KUKA KRL program: EPS_2_25716_MHDR05_A_20250926070358.src

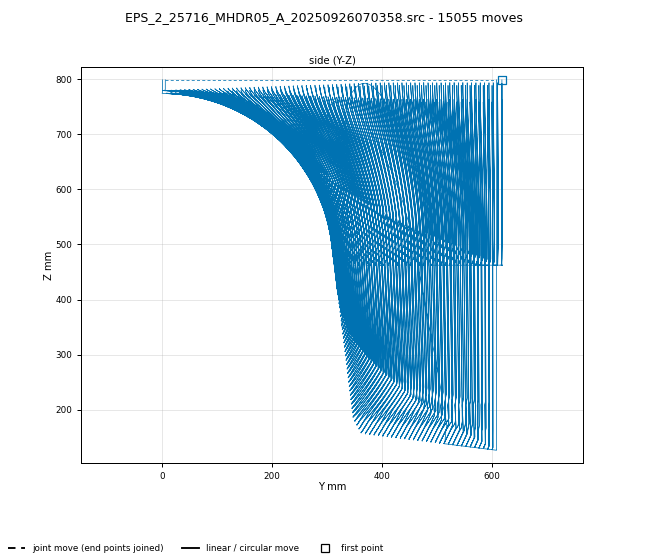
[picture p0: tool path of EPS_2_25716_MHDR05_A_20250926070358.src, 15055 of 15057 moves have a stored position in this frame; points joined in program order, loops and branches not executed]
&ACCESS RVP
&REL 4
&COMMENT QRS 19112012
&PARAM EDITMASK = *
DEF PART()
EXT BAS (BAS_COMMAND :IN,REAL :IN )
INT I
BAS (#INITMOV,0 )

;KUKA QRS Post kuka4.cps  Date:22-06-2017 !

File_ID=2854

QRS_PRE_INIT()

;Init var - Until changes are made in qrs_pre_init
Outlet_Square_prg=0
Inlet_1_Square_prg=0
Inlet_2_Square_prg=0
Inlet_3_Square_prg=0
Inlet_4_Square_prg=0
Inlet_5_Square_prg=0

Outlet_1={X 0.000, Y 400.000, Z 484.000, B 0.000, E1 0.000 }
Inlet_1={X 0.000, Y 425.000, Z 492.500, B 0.000, E1 180.000 }
Outlet_1_type=610
Inlet_1_type=533
;QRS#1=Sidecore dimensions
;QRS#2=600-24" Concrete
;QRS#3=525-21" Concrete
;QRS#4=
;QRS#5=
;QRS#6=
;QRS#7=
;QRS#8=
;QRS#9=S306-34L
;QRS#10=S306-32
;QRS#11=
;QRS#12=
;QRS#13=
;QRS#14=
;QRS#15=
;QRS#16=1220x127x1143 3,75'
;QRS#17=EPS Height
;QRS#18=789
;QRS#19=*
;QRS#20= UPDATED VERSION 22-06-2017
;QRS#21=*
Outlet_Square=0450
Inlet_1_Square=0250
Inlet_2_Square=0
Inlet_3_Square=0
Inlet_4_Square=0
Inlet_5_Square=0
Mill_Square=1
Outlet_Square_Prg=264
Inlet_1_Square_prg=263

QRS_INIT()

$ADVANCE=5

; T1
PTP {E1 171.039,E2 171.039}
PTP {X 0,Y 617.783,A -85,B 0,C 180,E1 171.039,E2 171.039,E3 0,E4 0,E5 0,E6 0}
QRS_SPEED_INIT()
LIN {X 0,Y 617.783,Z 799,A -85,B 0,C 180,E1 171.039,E2 171.039,E3 0,E4 0,E5 0,E6 0} C_VEL
LIN {X 0,Y 617.783,Z 464.44,A -85,B 0,C 180,E1 171.039,E2 171.039} C_VEL
LIN {X 0,Y 617.819,Z 462.44,A -85,B 0,C 180,E1 171.225,E2 171.225} C_VEL
LIN {X 0,Y 617.999,Z 462.44,A -85,B 0,C 180,E1 171.886,E2 171.886} C_VEL
LIN {X 0,Y 618.03,Z 462.44,A -85,B 0,C 180,E1 176.532,E2 176.532} C_VEL
LIN {X 0,Y 618.073,Z 462.44,A -85,B 0,C 180,E1 181.155,E2 181.155} C_VEL
LIN {X 0,Y 618.033,Z 462.44,A -85,B 0,C 180,E1 185.786,E2 185.786} C_VEL
LIN {X 0,Y 618.005,Z 462.44,A -85,B 0,C 180,E1 190.456,E2 190.456} C_VEL
LIN {X 0,Y 617.993,Z 462.44,A -85,B 0,C 180,E1 195.197,E2 195.197} C_VEL
LIN {X 0,Y 617.934,Z 462.44,A -85,B 0,C 180,E1 200.049,E2 200.049} C_VEL
LIN {X 0,Y 617.463,Z 462.44,A -85,B 0,C 180,E1 202.548,E2 202.548} C_VEL
LIN {X 0,Y 617.929,Z 462.44,A -85,B 0,C 180,E1 205.055,E2 205.055} C_VEL
LIN {X 0,Y 617.433,Z 462.44,A -85,B 0,C 180,E1 207.658,E2 207.658} C_VEL
LIN {X 0,Y 617.893,Z 462.44,A -85,B 0,C 180,E1 210.277,E2 210.277} C_VEL
LIN {X 0,Y 617.349,Z 462.44,A -85,B 0,C 180,E1 213.025,E2 213.025} C_VEL
LIN {X 0,Y 617.828,Z 462.44,A -85,B 0,C 180,E1 215.797,E2 215.797} C_VEL
LIN {X 0,Y 617.587,Z 462.44,A -85,B 0,C 180,E1 218.104,E2 218.104} C_VEL
LIN {X 0,Y 617.563,Z 462.44,A -85,B 0,C 180,E1 218.721,E2 218.721} C_VEL
LIN {X 0,Y 617.78,Z 462.44,A -85,B 0,C 180,E1 221.732,E2 221.732} C_VEL
LIN {X 0,Y 617.874,Z 462.44,A -85,B 0,C 180,E1 225.101,E2 225.101} C_VEL
LIN {X 0,Y 617.455,Z 462.44,A -85,B 0,C 180,E1 228.308,E2 228.308} C_VEL
LIN {X 0,Y 617.801,Z 462.44,A -85,B 0,C 180,E1 231.298,E2 231.298} C_VEL
LIN {X 0,Y 617.974,Z 462.44,A -85,B 0,C 180,E1 236.343,E2 236.343} C_VEL
LIN {X 0,Y 617.889,Z 462.44,A -85,B 0,C 180,E1 236.674,E2 236.674} C_VEL
LIN {X 0,Y 617.185,Z 462.44,A -85,B 0,C 180,E1 236.799,E2 236.799} C_VEL
LIN {X 0,Y 616.594,Z 462.517,A -85,B 0,C 180,E1 236.86,E2 236.86} C_VEL
LIN {X 0,Y 617.403,Z 470.086,A -85,B 0,C 180,E1 237.012,E2 237.012} C_VEL
LIN {X 0,Y 617.541,Z 504.624,A -85,B 0,C 180,E1 237.499,E2 237.499} C_VEL
LIN {X 0,Y 617.487,Z 514.142,A -85,B 0,C 180,E1 237.649,E2 237.649} C_VEL
LIN {X 0,Y 617.628,Z 530.885,A -85,B 0,C 180,E1 238.012,E2 238.012} C_VEL
LIN {X 0,Y 617.534,Z 541.25,A -85,B 0,C 180,E1 238.279,E2 238.279} C_VEL
LIN {X 0,Y 617.682,Z 548.357,A -85,B 0,C 180,E1 238.493,E2 238.493} C_VEL
LIN {X 0,Y 617.773,Z 561.084,A -85,B 0,C 180,E1 238.906,E2 238.906} C_VEL
LIN {X 0,Y 617.615,Z 577.198,A -85,B 0,C 180,E1 239.506,E2 239.506} C_VEL
LIN {X 0,Y 617.795,Z 590.272,A -85,B 0,C 180,E1 240.077,E2 240.077} C_VEL
LIN {X 0,Y 617.796,Z 604.603,A -85,B 0,C 180,E1 240.772,E2 240.772} C_VEL
LIN {X 0,Y 617.742,Z 616.6,A -85,B 0,C 180,E1 241.41,E2 241.41} C_VEL
LIN {X 0,Y 617.845,Z 630.486,A -85,B 0,C 180,E1 242.241,E2 242.241} C_VEL
LIN {X 0,Y 617.843,Z 644.637,A -85,B 0,C 180,E1 243.175,E2 243.175} C_VEL
LIN {X 0,Y 617.833,Z 656.904,A -85,B 0,C 180,E1 244.061,E2 244.061} C_VEL
LIN {X 0,Y 617.824,Z 668.121,A -85,B 0,C 180,E1 244.941,E2 244.941} C_VEL
LIN {X 0,Y 617.854,Z 679.212,A -85,B 0,C 180,E1 245.886,E2 245.886} C_VEL
LIN {X 0,Y 617.904,Z 690.179,A -85,B 0,C 180,E1 246.901,E2 246.901} C_VEL
LIN {X 0,Y 617.835,Z 700.537,A -85,B 0,C 180,E1 247.936,E2 247.936} C_VEL
LIN {X 0,Y 617.856,Z 710.526,A -85,B 0,C 180,E1 249.024,E2 249.024} C_VEL
LIN {X 0,Y 617.964,Z 719.897,A -85,B 0,C 180,E1 250.136,E2 250.136} C_VEL
LIN {X 0,Y 617.809,Z 728.454,A -85,B 0,C 180,E1 251.225,E2 251.225} C_VEL
LIN {X 0,Y 617.798,Z 736.799,A -85,B 0,C 180,E1 252.389,E2 252.389} C_VEL
LIN {X 0,Y 617.995,Z 744.741,A -85,B 0,C 180,E1 253.613,E2 253.613} C_VEL
LIN {X 0,Y 617.805,Z 751.886,A -85,B 0,C 180,E1 254.799,E2 254.799} C_VEL
LIN {X 0,Y 617.802,Z 759.815,A -85,B 0,C 180,E1 256.291,E2 256.291} C_VEL
LIN {X 0,Y 617.951,Z 765.481,A -85,B 0,C 180,E1 257.48,E2 257.48} C_VEL
LIN {X 0,Y 617.718,Z 771.737,A -85,B 0,C 180,E1 258.952,E2 258.952} C_VEL
LIN {X 0,Y 617.793,Z 776.648,A -85,B 0,C 180,E1 260.292,E2 260.292} C_VEL
LIN {X 0,Y 617.923,Z 780.377,A -85,B 0,C 180,E1 261.464,E2 261.464} C_VEL
LIN {X 0,Y 617.738,Z 784.109,A -85,B 0,C 180,E1 262.815,E2 262.815} C_VEL
LIN {X 0,Y 617.835,Z 787.205,A -85,B 0,C 180,E1 264.212,E2 264.212} C_VEL
LIN {X 0,Y 617.986,Z 788.8,A -85,B 0,C 180,E1 265.142,E2 265.142} C_VEL
LIN {X 0,Y 617.808,Z 790.277,A -85,B 0,C 180,E1 266.068,E2 266.068} C_VEL
LIN {X 0,Y 617.821,Z 792.139,A -85,B 0,C 180,E1 267.919,E2 267.919} C_VEL
LIN {X 0,Y 618.001,Z 792.641,A -85,B 0,C 180,E1 268.845,E2 268.845} C_VEL
LIN {X 0,Y 617.754,Z 792.708,A -85,B 0,C 180,E1 271.156,E2 271.156} C_VEL
LIN {X 0,Y 617.866,Z 792.126,A -85,B 0,C 180,E1 272.08,E2 272.08} C_VEL
LIN {X 0,Y 617.818,Z 790.825,A -85,B 0,C 180,E1 273.469,E2 273.469} C_VEL
LIN {X 0,Y 617.739,Z 789.656,A -85,B 0,C 180,E1 274.396,E2 274.396} C_VEL
LIN {X 0,Y 617.866,Z 787.197,A -85,B 0,C 180,E1 275.787,E2 275.787} C_VEL
LIN {X 0,Y 617.951,Z 785.135,A -85,B 0,C 180,E1 276.717,E2 276.717} C_VEL
LIN {X 0,Y 617.785,Z 782.833,A -85,B 0,C 180,E1 277.65,E2 277.65} C_VEL
LIN {X 0,Y 617.757,Z 779.54,A -85,B 0,C 180,E1 278.809,E2 278.809} C_VEL
LIN {X 0,Y 617.954,Z 775.427,A -85,B 0,C 180,E1 280.043,E2 280.043} C_VEL
LIN {X 0,Y 617.793,Z 770.565,A -85,B 0,C 180,E1 281.342,E2 281.342} C_VEL
LIN {X 0,Y 617.738,Z 765.525,A -85,B 0,C 180,E1 282.524,E2 282.524} C_VEL
LIN {X 0,Y 617.974,Z 758.301,A -85,B 0,C 180,E1 284.003,E2 284.003} C_VEL
LIN {X 0,Y 617.809,Z 750.854,A -85,B 0,C 180,E1 285.375,E2 285.375} C_VEL
LIN {X 0,Y 617.805,Z 743.014,A -85,B 0,C 180,E1 286.667,E2 286.667} C_VEL
LIN {X 0,Y 617.972,Z 735.018,A -85,B 0,C 180,E1 287.859,E2 287.859} C_VEL
LIN {X 0,Y 617.829,Z 726.926,A -85,B 0,C 180,E1 288.979,E2 288.979} C_VEL
LIN {X 0,Y 617.845,Z 717.147,A -85,B 0,C 180,E1 290.205,E2 290.205} C_VEL
LIN {X 0,Y 617.953,Z 707.77,A -85,B 0,C 180,E1 291.283,E2 291.283} C_VEL
LIN {X 0,Y 617.852,Z 697.496,A -85,B 0,C 180,E1 292.375,E2 292.375} C_VEL
LIN {X 0,Y 617.853,Z 687.7,A -85,B 0,C 180,E1 293.337,E2 293.337} C_VEL
LIN {X 0,Y 617.873,Z 676.158,A -85,B 0,C 180,E1 294.378,E2 294.378} C_VEL
LIN {X 0,Y 617.854,Z 665.151,A -85,B 0,C 180,E1 295.297,E2 295.297} C_VEL
LIN {X 0,Y 617.845,Z 652.567,A -85,B 0,C 180,E1 296.26,E2 296.26} C_VEL
LIN {X 0,Y 617.829,Z 641.105,A -85,B 0,C 180,E1 297.069,E2 297.069} C_VEL
LIN {X 0,Y 617.853,Z 627.693,A -85,B 0,C 180,E1 297.929,E2 297.929} C_VEL
LIN {X 0,Y 617.813,Z 613.836,A -85,B 0,C 180,E1 298.735,E2 298.735} C_VEL
LIN {X 0,Y 617.728,Z 602.666,A -85,B 0,C 180,E1 299.335,E2 299.335} C_VEL
LIN {X 0,Y 617.8,Z 586.176,A -85,B 0,C 180,E1 300.105,E2 300.105} C_VEL
LIN {X 0,Y 617.677,Z 572.126,A -85,B 0,C 180,E1 300.693,E2 300.693} C_VEL
LIN {X 0,Y 617.673,Z 563.857,A -85,B 0,C 180,E1 300.997,E2 300.997} C_VEL
LIN {X 0,Y 617.767,Z 554.861,A -85,B 0,C 180,E1 301.297,E2 301.297} C_VEL
LIN {X 0,Y 617.783,Z 545.131,A -85,B 0,C 180,E1 301.603,E2 301.603} C_VEL
LIN {X 0,Y 617.522,Z 529.56,A -85,B 0,C 180,E1 302.027,E2 302.027} C_VEL
LIN {X 0,Y 617.758,Z 515.151,A -85,B 0,C 180,E1 302.317,E2 302.317} C_VEL
LIN {X 0,Y 617.695,Z 494.179,A -85,B 0,C 180,E1 302.644,E2 302.644} C_VEL
LIN {X 0,Y 617.35,Z 469.361,A -85,B 0,C 180,E1 303.001,E2 303.001} C_VEL
LIN {X 0,Y 616.605,Z 462.44,A -85,B 0,C 180,E1 303.145,E2 303.145} C_VEL
LIN {X 0,Y 617.098,Z 462.44,A -85,B 0,C 180,E1 303.191,E2 303.191} C_VEL
LIN {X 0,Y 617.789,Z 462.44,A -85,B 0,C 180,E1 303.302,E2 303.302} C_VEL
LIN {X 0,Y 618.015,Z 462.44,A -85,B 0,C 180,E1 303.594,E2 303.594} C_VEL
LIN {X 0,Y 617.802,Z 462.44,A -85,B 0,C 180,E1 308.702,E2 308.702} C_VEL
LIN {X 0,Y 617.452,Z 462.44,A -85,B 0,C 180,E1 311.758,E2 311.758} C_VEL
LIN {X 0,Y 617.87,Z 462.44,A -85,B 0,C 180,E1 314.9,E2 314.9} C_VEL
LIN {X 0,Y 617.779,Z 462.44,A -85,B 0,C 180,E1 318.272,E2 318.272} C_VEL
LIN {X 0,Y 617.56,Z 462.44,A -85,B 0,C 180,E1 321.279,E2 321.279} C_VEL
LIN {X 0,Y 617.589,Z 462.44,A -85,B 0,C 180,E1 321.896,E2 321.896} C_VEL
LIN {X 0,Y 617.821,Z 462.44,A -85,B 0,C 180,E1 324.202,E2 324.202} C_VEL
LIN {X 0,Y 617.351,Z 462.44,A -85,B 0,C 180,E1 326.975,E2 326.975} C_VEL
LIN {X 0,Y 617.885,Z 462.44,A -85,B 0,C 180,E1 329.722,E2 329.722} C_VEL
LIN {X 0,Y 617.419,Z 462.44,A -85,B 0,C 180,E1 332.341,E2 332.341} C_VEL
LIN {X 0,Y 617.911,Z 462.44,A -85,B 0,C 180,E1 334.944,E2 334.944} C_VEL
LIN {X 0,Y 617.452,Z 462.44,A -85,B 0,C 180,E1 337.452,E2 337.452} C_VEL
LIN {X 0,Y 617.95,Z 462.44,A -85,B 0,C 180,E1 339.951,E2 339.951} C_VEL
LIN {X 0,Y 618.038,Z 462.44,A -85,B 0,C 180,E1 343.627,E2 343.627} C_VEL
LIN {X 0,Y 617.996,Z 462.44,A -85,B 0,C 180,E1 349.544,E2 349.544} C_VEL
LIN {X 0,Y 618.025,Z 462.44,A -85,B 0,C 180,E1 354.214,E2 354.214} C_VEL
LIN {X 0,Y 618.072,Z 462.44,A -85,B 0,C 180,E1 358.845,E2 358.845} C_VEL
LIN {X 0,Y 618.015,Z 462.44,A -85,B 0,C 180,E1 363.468,E2 363.468} C_VEL
LIN {X 0,Y 618.004,Z 462.44,A -85,B 0,C 180,E1 368.114,E2 368.114} C_VEL
LIN {X 0,Y 617.996,Z 462.44,A -85,B 0,C 180,E1 372.815,E2 372.815} C_VEL
LIN {X 0,Y 617.929,Z 462.44,A -85,B 0,C 180,E1 377.608,E2 377.608} C_VEL
LIN {X 0,Y 617.74,Z 462.44,A -85,B 0,C 180,E1 378.544,E2 378.544} C_VEL
LIN {X 0,Y 617.922,Z 462.44,A -85,B 0,C 180,E1 382.53,E2 382.53} C_VEL
LIN {X 0,Y 617.417,Z 462.44,A -85,B 0,C 180,E1 385.078,E2 385.078} C_VEL
LIN {X 0,Y 617.852,Z 462.44,A -85,B 0,C 180,E1 387.638,E2 387.638} C_VEL
LIN {X 0,Y 617.402,Z 462.44,A -85,B 0,C 180,E1 390.304,E2 390.304} C_VEL
LIN {X 0,Y 617.942,Z 462.44,A -85,B 0,C 180,E1 392.989,E2 392.989} C_VEL
LIN {X 0,Y 617.669,Z 462.44,A -85,B 0,C 180,E1 395.808,E2 395.808} C_VEL
LIN {X 0,Y 617.67,Z 462.44,A -85,B 0,C 180,E1 398.113,E2 398.113} C_VEL
LIN {X 0,Y 617.779,Z 462.44,A -85,B 0,C 180,E1 401.732,E2 401.732} C_VEL
LIN {X 0,Y 617.379,Z 462.44,A -85,B 0,C 180,E1 405.055,E2 405.055} C_VEL
LIN {X 0,Y 617.751,Z 462.44,A -85,B 0,C 180,E1 408.277,E2 408.277} C_VEL
LIN {X 0,Y 617.719,Z 462.44,A -85,B 0,C 180,E1 411.883,E2 411.883} C_VEL
LIN {X 0,Y 617.766,Z 462.44,A -85,B 0,C 180,E1 414.2,E2 414.2} C_VEL
LIN {X 0,Y 617.866,Z 462.44,A -85,B 0,C 180,E1 415.782,E2 415.782} C_VEL
LIN {X 0,Y 617.926,Z 462.44,A -85,B 0,C 180,E1 417.011,E2 417.011} C_VEL
LIN {X 0,Y 618.067,Z 462.44,A -85,B 0,C 180,E1 420.693,E2 420.693} C_VEL
LIN {X 0,Y 616.955,Z 462.44,A -85,B 0,C 180,E1 420.924,E2 420.924} C_VEL
LIN {X 0,Y 617.604,Z 503.778,A -85,B 0,C 180,E1 421.5,E2 421.5} C_VEL
LIN {X 0,Y 617.775,Z 519.441,A -85,B 0,C 180,E1 421.761,E2 421.761} C_VEL
LIN {X 0,Y 617.726,Z 532.784,A -85,B 0,C 180,E1 422.041,E2 422.041} C_VEL
LIN {X 0,Y 617.742,Z 541.12,A -85,B 0,C 180,E1 422.253,E2 422.253} C_VEL
LIN {X 0,Y 617.897,Z 557,A -85,B 0,C 180,E1 422.731,E2 422.731} C_VEL
LIN {X 0,Y 617.825,Z 571.564,A -85,B 0,C 180,E1 423.255,E2 423.255} C_VEL
LIN {X 0,Y 617.785,Z 579.5,A -85,B 0,C 180,E1 423.576,E2 423.576} C_VEL
LIN {X 0,Y 617.917,Z 593.777,A -85,B 0,C 180,E1 424.225,E2 424.225} C_VEL
LIN {X 0,Y 617.894,Z 607.704,A -85,B 0,C 180,E1 424.944,E2 424.944} C_VEL
LIN {X 0,Y 617.898,Z 620.167,A -85,B 0,C 180,E1 425.668,E2 425.668} C_VEL
LIN {X 0,Y 617.917,Z 631.689,A -85,B 0,C 180,E1 426.409,E2 426.409} C_VEL
LIN {X 0,Y 617.928,Z 642.528,A -85,B 0,C 180,E1 427.172,E2 427.172} C_VEL
LIN {X 0,Y 617.917,Z 652.557,A -85,B 0,C 180,E1 427.939,E2 427.939} C_VEL
LIN {X 0,Y 617.883,Z 663.654,A -85,B 0,C 180,E1 428.87,E2 428.87} C_VEL
LIN {X 0,Y 617.918,Z 672.158,A -85,B 0,C 180,E1 429.643,E2 429.643} C_VEL
LIN {X 0,Y 617.951,Z 680.759,A -85,B 0,C 180,E1 430.489,E2 430.489} C_VEL
LIN {X 0,Y 617.882,Z 689.526,A -85,B 0,C 180,E1 431.422,E2 431.422} C_VEL
LIN {X 0,Y 617.893,Z 697.879,A -85,B 0,C 180,E1 432.392,E2 432.392} C_VEL
LIN {X 0,Y 617.964,Z 706.601,A -85,B 0,C 180,E1 433.508,E2 433.508} C_VEL
LIN {X 0,Y 617.846,Z 714.508,A -85,B 0,C 180,E1 434.611,E2 434.611} C_VEL
LIN {X 0,Y 617.865,Z 719.734,A -85,B 0,C 180,E1 435.398,E2 435.398} C_VEL
LIN {X 0,Y 617.957,Z 726.877,A -85,B 0,C 180,E1 436.591,E2 436.591} C_VEL
LIN {X 0,Y 617.781,Z 733.283,A -85,B 0,C 180,E1 437.773,E2 437.773} C_VEL
LIN {X 0,Y 617.815,Z 738.937,A -85,B 0,C 180,E1 438.953,E2 438.953} C_VEL
LIN {X 0,Y 617.968,Z 743.151,A -85,B 0,C 180,E1 439.948,E2 439.948} C_VEL
LIN {X 0,Y 617.808,Z 748.098,A -85,B 0,C 180,E1 441.244,E2 441.244} C_VEL
LIN {X 0,Y 617.809,Z 751.662,A -85,B 0,C 180,E1 442.35,E2 442.35} C_VEL
LIN {X 0,Y 617.965,Z 755.451,A -85,B 0,C 180,E1 443.749,E2 443.749} C_VEL
LIN {X 0,Y 617.799,Z 757.522,A -85,B 0,C 180,E1 444.676,E2 444.676} C_VEL
LIN {X 0,Y 617.741,Z 759.253,A -85,B 0,C 180,E1 445.604,E2 445.604} C_VEL
LIN {X 0,Y 617.829,Z 760.65,A -85,B 0,C 180,E1 446.531,E2 446.531} C_VEL
LIN {X 0,Y 617.883,Z 762.082,A -85,B 0,C 180,E1 447.92,E2 447.92} C_VEL
LIN {X 0,Y 617.759,Z 762.722,A -85,B 0,C 180,E1 448.844,E2 448.844} C_VEL
LIN {X 0,Y 617.984,Z 762.639,A -85,B 0,C 180,E1 451.155,E2 451.155} C_VEL
LIN {X 0,Y 617.844,Z 762.029,A -85,B 0,C 180,E1 452.08,E2 452.08} C_VEL
LIN {X 0,Y 617.811,Z 760.549,A -85,B 0,C 180,E1 453.469,E2 453.469} C_VEL
LIN {X 0,Y 617.968,Z 758.269,A -85,B 0,C 180,E1 454.858,E2 454.858} C_VEL
LIN {X 0,Y 617.795,Z 755.261,A -85,B 0,C 180,E1 456.253,E2 456.253} C_VEL
LIN {X 0,Y 617.901,Z 751.349,A -85,B 0,C 180,E1 457.649,E2 457.649} C_VEL
LIN {X 0,Y 617.95,Z 748.595,A -85,B 0,C 180,E1 458.504,E2 458.504} C_VEL
LIN {X 0,Y 617.786,Z 744.33,A -85,B 0,C 180,E1 459.676,E2 459.676} C_VEL
LIN {X 0,Y 617.873,Z 738.532,A -85,B 0,C 180,E1 461.046,E2 461.046} C_VEL
LIN {X 0,Y 617.956,Z 734.237,A -85,B 0,C 180,E1 461.928,E2 461.928} C_VEL
LIN {X 0,Y 617.877,Z 731.217,A -85,B 0,C 180,E1 462.521,E2 462.521} C_VEL
LIN {X 0,Y 617.813,Z 726.388,A -85,B 0,C 180,E1 463.412,E2 463.412} C_VEL
LIN {X 0,Y 617.915,Z 719.127,A -85,B 0,C 180,E1 464.6,E2 464.6} C_VEL
LIN {X 0,Y 617.914,Z 711.371,A -85,B 0,C 180,E1 465.75,E2 465.75} C_VEL
LIN {X 0,Y 617.856,Z 703.85,A -85,B 0,C 180,E1 466.77,E2 466.77} C_VEL
LIN {X 0,Y 617.955,Z 696.029,A -85,B 0,C 180,E1 467.736,E2 467.736} C_VEL
LIN {X 0,Y 617.947,Z 688.072,A -85,B 0,C 180,E1 468.646,E2 468.646} C_VEL
LIN {X 0,Y 617.889,Z 677.993,A -85,B 0,C 180,E1 469.698,E2 469.698} C_VEL
LIN {X 0,Y 617.935,Z 669.53,A -85,B 0,C 180,E1 470.51,E2 470.51} C_VEL
LIN {X 0,Y 617.943,Z 660.871,A -85,B 0,C 180,E1 471.283,E2 471.283} C_VEL
LIN {X 0,Y 617.897,Z 649.404,A -85,B 0,C 180,E1 472.218,E2 472.218} C_VEL
LIN {X 0,Y 617.901,Z 639.435,A -85,B 0,C 180,E1 472.964,E2 472.964} C_VEL
LIN {X 0,Y 617.901,Z 627.869,A -85,B 0,C 180,E1 473.754,E2 473.754} C_VEL
LIN {X 0,Y 617.908,Z 616.74,A -85,B 0,C 180,E1 474.447,E2 474.447} C_VEL
LIN {X 0,Y 617.878,Z 604.518,A -85,B 0,C 180,E1 475.136,E2 475.136} C_VEL
LIN {X 0,Y 617.817,Z 593.563,A -85,B 0,C 180,E1 475.699,E2 475.699} C_VEL
LIN {X 0,Y 617.912,Z 581.251,A -85,B 0,C 180,E1 476.257,E2 476.257} C_VEL
LIN {X 0,Y 617.845,Z 567.047,A -85,B 0,C 180,E1 476.825,E2 476.825} C_VEL
LIN {X 0,Y 617.714,Z 555.11,A -85,B 0,C 180,E1 477.247,E2 477.247} C_VEL
LIN {X 0,Y 617.848,Z 541.717,A -85,B 0,C 180,E1 477.637,E2 477.637} C_VEL
LIN {X 0,Y 617.777,Z 527.547,A -85,B 0,C 180,E1 477.985,E2 477.985} C_VEL
LIN {X 0,Y 617.682,Z 517.241,A -85,B 0,C 180,E1 478.198,E2 478.198} C_VEL
LIN {X 0,Y 617.703,Z 498.206,A -85,B 0,C 180,E1 478.478,E2 478.478} C_VEL
LIN {X 0,Y 617.585,Z 474.624,A -85,B 0,C 180,E1 478.79,E2 478.79} C_VEL
LIN {X 0,Y 616.866,Z 466.499,A -85,B 0,C 180,E1 478.932,E2 478.932} C_VEL
LIN {X 0,Y 616.534,Z 463.909,A -85,B 0,C 180,E1 478.983,E2 478.983} C_VEL
LIN {X 0,Y 616.608,Z 462.44,A -85,B 0,C 180,E1 479.035,E2 479.035} C_VEL
LIN {X 0,Y 616.994,Z 462.44,A -85,B 0,C 180,E1 479.071,E2 479.071} C_VEL
LIN {X 0,Y 617.992,Z 462.44,A -85,B 0,C 180,E1 479.266,E2 479.266} C_VEL
LIN {X 0,Y 618.022,Z 462.44,A -85,B 0,C 180,E1 480.269,E2 480.269} C_VEL
LIN {X 0,Y 617.371,Z 462.44,A -85,B 0,C 180,E1 484.15,E2 484.15} C_VEL
LIN {X 0,Y 617.837,Z 462.44,A -85,B 0,C 180,E1 485.795,E2 485.795} C_VEL
LIN {X 0,Y 617.917,Z 462.44,A -85,B 0,C 180,E1 488.693,E2 488.693} C_VEL
LIN {X 0,Y 617.4,Z 462.44,A -85,B 0,C 180,E1 491.762,E2 491.762} C_VEL
LIN {X 0,Y 617.798,Z 462.44,A -85,B 0,C 180,E1 494.906,E2 494.906} C_VEL
LIN {X 0,Y 617.752,Z 462.44,A -85,B 0,C 180,E1 498.275,E2 498.275} C_VEL
LIN {X 0,Y 617.543,Z 462.44,A -85,B 0,C 180,E1 501.278,E2 501.278} C_VEL
LIN {X 0,Y 617.803,Z 462.44,A -85,B 0,C 180,E1 504.201,E2 504.201} C_VEL
LIN {X 0,Y 617.344,Z 462.44,A -85,B 0,C 180,E1 506.975,E2 506.975} C_VEL
LIN {X 0,Y 617.901,Z 462.44,A -85,B 0,C 180,E1 509.723,E2 509.723} C_VEL
LIN {X 0,Y 617.406,Z 462.44,A -85,B 0,C 180,E1 512.34,E2 512.34} C_VEL
LIN {X 0,Y 617.873,Z 462.44,A -85,B 0,C 180,E1 514.942,E2 514.942} C_VEL
LIN {X 0,Y 617.432,Z 462.44,A -85,B 0,C 180,E1 517.451,E2 517.451} C_VEL
LIN {X 0,Y 617.948,Z 462.44,A -85,B 0,C 180,E1 519.951,E2 519.951} C_VEL
LIN {X 0,Y 617.722,Z 462.44,A -85,B 0,C 180,E1 522.386,E2 522.386} C_VEL
LIN {X 0,Y 617.816,Z 462.44,A -85,B 0,C 180,E1 524.799,E2 524.799} C_VEL
LIN {X 0,Y 618.009,Z 462.44,A -85,B 0,C 180,E1 527.185,E2 527.185} C_VEL
LIN {X 0,Y 617.819,Z 462.44,A -85,B 0,C 180,E1 531.225,E2 531.225} C_VEL
LIN {X 0,Y 615.297,Z 462.44,A -85,B 0,C 180,E1 532.421,E2 532.421} C_VEL
LIN {X 0,Y 609.713,Z 462.44,A -85,B 0,C 180,E1 534.209,E2 534.209} C_VEL
LIN {X 0,Y 609.626,Z 462.44,A -85,B 0,C 180,E1 534.416,E2 534.416} C_VEL
LIN {X 0,Y 609.654,Z 462.44,A -85,B 0,C 180,E1 538.578,E2 538.578} C_VEL
LIN {X 0,Y 609.702,Z 462.44,A -85,B 0,C 180,E1 542.847,E2 542.847} C_VEL
LIN {X 0,Y 609.732,Z 462.44,A -85,B 0,C 180,E1 547.132,E2 547.132} C_VEL
LIN {X 0,Y 609.776,Z 462.44,A -85,B 0,C 180,E1 551.457,E2 551.457} C_VEL
LIN {X 0,Y 609.824,Z 462.44,A -85,B 0,C 180,E1 555.849,E2 555.849} C_VEL
LIN {X 0,Y 609.947,Z 462.44,A -85,B 0,C 180,E1 560.335,E2 560.335} C_VEL
LIN {X 0,Y 610.013,Z 462.44,A -85,B 0,C 180,E1 564.956,E2 564.956} C_VEL
LIN {X 0,Y 609.819,Z 462.44,A -85,B 0,C 180,E1 569.771,E2 569.771} C_VEL
LIN {X 0,Y 609.765,Z 462.44,A -85,B 0,C 180,E1 576.577,E2 576.577} C_VEL
LIN {X 0,Y 609.787,Z 462.44,A -85,B 0,C 180,E1 582.095,E2 582.095} C_VEL
LIN {X 0,Y 609.499,Z 462.44,A -85,B 0,C 180,E1 587.876,E2 587.876} C_VEL
LIN {X 0,Y 609.495,Z 462.44,A -85,B 0,C 180,E1 592.644,E2 592.644} C_VEL
LIN {X 0,Y 610.021,Z 462.44,A -85,B 0,C 180,E1 596.454,E2 596.454} C_VEL
LIN {X 0,Y 610.903,Z 528.821,A -85,B 0,C 180,E1 597.568,E2 597.568} C_VEL
LIN {X 0,Y 610.845,Z 569.805,A -85,B 0,C 180,E1 598.839,E2 598.839} C_VEL
LIN {X 0,Y 610.681,Z 607.941,A -85,B 0,C 180,E1 600.578,E2 600.578} C_VEL
LIN {X 0,Y 610.557,Z 644.898,A -85,B 0,C 180,E1 602.847,E2 602.847} C_VEL
LIN {X 0,Y 610.358,Z 679.993,A -85,B 0,C 180,E1 605.643,E2 605.643} C_VEL
LIN {X 0,Y 610.195,Z 711.949,A -85,B 0,C 180,E1 608.912,E2 608.912} C_VEL
LIN {X 0,Y 610.056,Z 737.919,A -85,B 0,C 180,E1 612.3,E2 612.3} C_VEL
LIN {X 0,Y 610.002,Z 759.715,A -85,B 0,C 180,E1 615.995,E2 615.995} C_VEL
LIN {X 0,Y 609.93,Z 775.429,A -85,B 0,C 180,E1 619.631,E2 619.631} C_VEL
LIN {X 0,Y 609.923,Z 785.996,A -85,B 0,C 180,E1 623.165,E2 623.165} C_VEL
LIN {X 0,Y 610.059,Z 790.904,A -85,B 0,C 180,E1 625.73,E2 625.73} C_VEL
LIN {X 0,Y 610.125,Z 793.656,A -85,B 0,C 180,E1 628.578,E2 628.578} C_VEL
LIN {X 0,Y 610.01,Z 792.627,A -85,B 0,C 180,E1 632.845,E2 632.845} C_VEL
LIN {X 0,Y 610.071,Z 785.331,A -85,B 0,C 180,E1 637.128,E2 637.128} C_VEL
LIN {X 0,Y 609.997,Z 772.733,A -85,B 0,C 180,E1 641.091,E2 641.091} C_VEL
LIN {X 0,Y 610.035,Z 754.01,A -85,B 0,C 180,E1 645.071,E2 645.071} C_VEL
LIN {X 0,Y 610.148,Z 731.347,A -85,B 0,C 180,E1 648.633,E2 648.633} C_VEL
LIN {X 0,Y 610.269,Z 703.401,A -85,B 0,C 180,E1 652.041,E2 652.041} C_VEL
LIN {X 0,Y 610.395,Z 671.004,A -85,B 0,C 180,E1 655.138,E2 655.138} C_VEL
LIN {X 0,Y 610.619,Z 634.981,A -85,B 0,C 180,E1 657.819,E2 657.819} C_VEL
LIN {X 0,Y 610.736,Z 597.02,A -85,B 0,C 180,E1 659.978,E2 659.978} C_VEL
LIN {X 0,Y 610.944,Z 558.595,A -85,B 0,C 180,E1 661.568,E2 661.568} C_VEL
LIN {X 0,Y 610.989,Z 519.348,A -85,B 0,C 180,E1 662.63,E2 662.63} C_VEL
LIN {X 0,Y 610.007,Z 462.44,A -85,B 0,C 180,E1 663.548,E2 663.548} C_VEL
LIN {X 0,Y 609.604,Z 462.44,A -85,B 0,C 180,E1 669.655,E2 669.655} C_VEL
LIN {X 0,Y 609.725,Z 462.44,A -85,B 0,C 180,E1 675.952,E2 675.952} C_VEL
LIN {X 0,Y 609.565,Z 462.44,A -85,B 0,C 180,E1 680.356,E2 680.356} C_VEL
LIN {X 0,Y 609.614,Z 462.44,A -85,B 0,C 180,E1 685.165,E2 685.165} C_VEL
LIN {X 0,Y 609.752,Z 462.44,A -85,B 0,C 180,E1 690.356,E2 690.356} C_VEL
LIN {X 0,Y 609.986,Z 462.44,A -85,B 0,C 180,E1 695.043,E2 695.043} C_VEL
LIN {X 0,Y 609.8,Z 462.44,A -85,B 0,C 180,E1 701.17,E2 701.17} C_VEL
LIN {X 0,Y 609.372,Z 462.44,A -85,B 0,C 180,E1 705.708,E2 705.708} C_VEL
LIN {X 0,Y 609.93,Z 462.44,A -85,B 0,C 180,E1 709.993,E2 709.993} C_VEL
LIN {X 0,Y 610.105,Z 462.44,A -85,B 0,C 180,E1 714.303,E2 714.303} C_VEL
LIN {X 0,Y 609.785,Z 462.44,A -85,B 0,C 180,E1 719.999,E2 719.999} C_VEL
LIN {X 0,Y 609.821,Z 462.44,A -85,B 0,C 180,E1 724.27,E2 724.27} C_VEL
LIN {X 0,Y 609.939,Z 462.44,A -85,B 0,C 180,E1 728.564,E2 728.564} C_VEL
LIN {X 0,Y 610.049,Z 462.44,A -85,B 0,C 180,E1 732.905,E2 732.905} C_VEL
LIN {X 0,Y 609.752,Z 462.44,A -85,B 0,C 180,E1 738.83,E2 738.83} C_VEL
LIN {X 0,Y 609.723,Z 462.44,A -85,B 0,C 180,E1 743.408,E2 743.408} C_VEL
LIN {X 0,Y 609.772,Z 462.44,A -85,B 0,C 180,E1 748.146,E2 748.146} C_VEL
LIN {X 0,Y 610.002,Z 462.44,A -85,B 0,C 180,E1 753.093,E2 753.093} C_VEL
LIN {X 0,Y 609.71,Z 462.44,A -85,B 0,C 180,E1 758.371,E2 758.371} C_VEL
LIN {X 0,Y 609.751,Z 462.44,A -85,B 0,C 180,E1 762.096,E2 762.096} C_VEL
LIN {X 0,Y 609.815,Z 462.44,A -85,B 0,C 180,E1 768.14,E2 768.14} C_VEL
LIN {X 0,Y 609.757,Z 462.44,A -85,B 0,C 180,E1 773.419,E2 773.419} C_VEL
LIN {X 0,Y 609.801,Z 462.44,A -85,B 0,C 180,E1 778.572,E2 778.572} C_VEL
LIN {X 0,Y 610.106,Z 462.44,A -85,B 0,C 180,E1 780.548,E2 780.548} C_VEL
LIN {X 0,Y 610.781,Z 530.926,A -85,B 0,C 180,E1 781.648,E2 781.648} C_VEL
LIN {X 0,Y 610.682,Z 571.82,A -85,B 0,C 180,E1 782.928,E2 782.928} C_VEL
LIN {X 0,Y 610.554,Z 610.259,A -85,B 0,C 180,E1 784.771,E2 784.771} C_VEL
LIN {X 0,Y 610.419,Z 645.444,A -85,B 0,C 180,E1 787.1,E2 787.1} C_VEL
LIN {X 0,Y 610.269,Z 676.426,A -85,B 0,C 180,E1 789.797,E2 789.797} C_VEL
LIN {X 0,Y 610.184,Z 703.547,A -85,B 0,C 180,E1 792.862,E2 792.862} C_VEL
LIN {X 0,Y 610.158,Z 727.018,A -85,B 0,C 180,E1 796.364,E2 796.364} C_VEL
LIN {X 0,Y 610.141,Z 744.589,A -85,B 0,C 180,E1 799.996,E2 799.996} C_VEL
LIN {X 0,Y 610.136,Z 756.155,A -85,B 0,C 180,E1 803.588,E2 803.588} C_VEL
LIN {X 0,Y 609.994,Z 762.448,A -85,B 0,C 180,E1 807.154,E2 807.154} C_VEL
LIN {X 0,Y 609.963,Z 763.996,A -85,B 0,C 180,E1 810,E2 810} C_VEL
LIN {X 0,Y 609.962,Z 762.34,A -85,B 0,C 180,E1 812.846,E2 812.846} C_VEL
LIN {X 0,Y 609.981,Z 755.913,A -85,B 0,C 180,E1 816.414,E2 816.414} C_VEL
LIN {X 0,Y 609.97,Z 744.214,A -85,B 0,C 180,E1 820.007,E2 820.007} C_VEL
LIN {X 0,Y 610.042,Z 727.556,A -85,B 0,C 180,E1 823.455,E2 823.455} C_VEL
LIN {X 0,Y 610.144,Z 704.305,A -85,B 0,C 180,E1 826.953,E2 826.953} C_VEL
LIN {X 0,Y 610.249,Z 676.792,A -85,B 0,C 180,E1 830.077,E2 830.077} C_VEL
LIN {X 0,Y 610.412,Z 645.526,A -85,B 0,C 180,E1 832.804,E2 832.804} C_VEL
LIN {X 0,Y 610.56,Z 612.081,A -85,B 0,C 180,E1 835.033,E2 835.033} C_VEL
LIN {X 0,Y 610.723,Z 575.633,A -85,B 0,C 180,E1 836.823,E2 836.823} C_VEL
LIN {X 0,Y 610.826,Z 540.974,A -85,B 0,C 180,E1 838.002,E2 838.002} C_VEL
LIN {X 0,Y 610.802,Z 503.888,A -85,B 0,C 180,E1 838.755,E2 838.755} C_VEL
LIN {X 0,Y 609.67,Z 465.143,A -85,B 0,C 180,E1 839.326,E2 839.326} C_VEL
LIN {X 0,Y 609.946,Z 462.44,A -85,B 0,C 180,E1 839.43,E2 839.43} C_VEL
LIN {X 0,Y 609.805,Z 462.44,A -85,B 0,C 180,E1 846.578,E2 846.578} C_VEL
LIN {X 0,Y 609.536,Z 462.44,A -85,B 0,C 180,E1 850.23,E2 850.23} C_VEL
LIN {X 0,Y 609.646,Z 462.44,A -85,B 0,C 180,E1 856.075,E2 856.075} C_VEL
LIN {X 0,Y 609.528,Z 462.44,A -85,B 0,C 180,E1 860.361,E2 860.361} C_VEL
LIN {X 0,Y 609.595,Z 462.44,A -85,B 0,C 180,E1 865.166,E2 865.166} C_VEL
LIN {X 0,Y 609.772,Z 462.44,A -85,B 0,C 180,E1 870.353,E2 870.353} C_VEL
LIN {X 0,Y 609.96,Z 462.44,A -85,B 0,C 180,E1 875.043,E2 875.043} C_VEL
LIN {X 0,Y 609.825,Z 462.44,A -85,B 0,C 180,E1 881.172,E2 881.172} C_VEL
LIN {X 0,Y 610.097,Z 462.44,A -85,B 0,C 180,E1 887.096,E2 887.096} C_VEL
LIN {X 0,Y 609.775,Z 462.44,A -85,B 0,C 180,E1 892.87,E2 892.87} C_VEL
LIN {X 0,Y 609.626,Z 462.44,A -85,B 0,C 180,E1 894.416,E2 894.416} C_VEL
LIN {X 0,Y 605.866,Z 462.44,A -85,B 0,C 180,E1 896.023,E2 896.023} C_VEL
LIN {X 0,Y 601.872,Z 462.44,A -85,B 0,C 180,E1 897.65,E2 897.65} C_VEL
LIN {X 0,Y 602.167,Z 462.44,A -85,B 0,C 180,E1 901.441,E2 901.441} C_VEL
LIN {X 0,Y 602.186,Z 462.44,A -85,B 0,C 180,E1 905.772,E2 905.772} C_VEL
LIN {X 0,Y 601.857,Z 462.44,A -85,B 0,C 180,E1 911.61,E2 911.61} C_VEL
LIN {X 0,Y 601.855,Z 462.44,A -85,B 0,C 180,E1 916.064,E2 916.064} C_VEL
LIN {X 0,Y 601.746,Z 462.44,A -85,B 0,C 180,E1 921.408,E2 921.408} C_VEL
LIN {X 0,Y 601.988,Z 462.44,A -85,B 0,C 180,E1 925.312,E2 925.312} C_VEL
LIN {X 0,Y 601.722,Z 462.44,A -85,B 0,C 180,E1 931.179,E2 931.179} C_VEL
LIN {X 0,Y 601.787,Z 462.44,A -85,B 0,C 180,E1 937.142,E2 937.142} C_VEL
LIN {X 0,Y 601.772,Z 462.44,A -85,B 0,C 180,E1 943.141,E2 943.141} C_VEL
LIN {X 0,Y 601.576,Z 462.44,A -85,B 0,C 180,E1 949.125,E2 949.125} C_VEL
LIN {X 0,Y 601.504,Z 462.44,A -85,B 0,C 180,E1 953.652,E2 953.652} C_VEL
LIN {X 0,Y 601.989,Z 462.44,A -85,B 0,C 180,E1 955.936,E2 955.936} C_VEL
LIN {X 0,Y 604.143,Z 471.909,A -85,B 0,C 180,E1 956.217,E2 956.217} C_VEL
LIN {X 0,Y 604.193,Z 527.758,A -85,B 0,C 180,E1 957.14,E2 957.14} C_VEL
LIN {X 0,Y 604.024,Z 565.871,A -85,B 0,C 180,E1 958.298,E2 958.298} C_VEL
LIN {X 0,Y 603.692,Z 605.048,A -85,B 0,C 180,E1 960.044,E2 960.044} C_VEL
LIN {X 0,Y 603.333,Z 642.732,A -85,B 0,C 180,E1 962.336,E2 962.336} C_VEL
LIN {X 0,Y 602.867,Z 679.987,A -85,B 0,C 180,E1 965.32,E2 965.32} C_VEL
LIN {X 0,Y 602.533,Z 711.01,A -85,B 0,C 180,E1 968.518,E2 968.518} C_VEL
LIN {X 0,Y 602.265,Z 737.921,A -85,B 0,C 180,E1 972.063,E2 972.063} C_VEL
LIN {X 0,Y 602.157,Z 759.715,A -85,B 0,C 180,E1 975.808,E2 975.808} C_VEL
LIN {X 0,Y 602.051,Z 775.739,A -85,B 0,C 180,E1 979.578,E2 979.578} C_VEL
LIN {X 0,Y 602.027,Z 785.331,A -85,B 0,C 180,E1 982.776,E2 982.776} C_VEL
LIN {X 0,Y 602.18,Z 790.904,A -85,B 0,C 180,E1 985.674,E2 985.674} C_VEL
LIN {X 0,Y 602.219,Z 793.657,A -85,B 0,C 180,E1 988.559,E2 988.559} C_VEL
LIN {X 0,Y 602.104,Z 792.627,A -85,B 0,C 180,E1 992.883,E2 992.883} C_VEL
LIN {X 0,Y 602.193,Z 786.221,A -85,B 0,C 180,E1 996.818,E2 996.818} C_VEL
LIN {X 0,Y 602.165,Z 774.656,A -85,B 0,C 180,E1 1000.714,E2 1000.714} C_VEL
LIN {X 0,Y 602.258,Z 757.765,A -85,B 0,C 180,E1 1004.561,E2 1004.561} C_VEL
LIN {X 0,Y 602.417,Z 735.374,A -85,B 0,C 180,E1 1008.311,E2 1008.311} C_VEL
LIN {X 0,Y 602.661,Z 708.058,A -85,B 0,C 180,E1 1011.82,E2 1011.82} C_VEL
LIN {X 0,Y 602.935,Z 676.292,A -85,B 0,C 180,E1 1015.011,E2 1015.011} C_VEL
LIN {X 0,Y 603.346,Z 639.736,A -85,B 0,C 180,E1 1017.866,E2 1017.866} C_VEL
LIN {X 0,Y 603.706,Z 600.519,A -85,B 0,C 180,E1 1020.192,E2 1020.192} C_VEL
LIN {X 0,Y 604.136,Z 559.476,A -85,B 0,C 180,E1 1021.937,E2 1021.937} C_VEL
LIN {X 0,Y 604.327,Z 519.965,A -85,B 0,C 180,E1 1023.022,E2 1023.022} C_VEL
LIN {X 0,Y 603.396,Z 466.841,A -85,B 0,C 180,E1 1023.901,E2 1023.901} C_VEL
LIN {X 0,Y 601.975,Z 462.44,A -85,B 0,C 180,E1 1024.106,E2 1024.106} C_VEL
LIN {X 0,Y 601.769,Z 462.44,A -85,B 0,C 180,E1 1028.979,E2 1028.979} C_VEL
LIN {X 0,Y 601.728,Z 462.44,A -85,B 0,C 180,E1 1035.211,E2 1035.211} C_VEL
LIN {X 0,Y 601.718,Z 462.44,A -85,B 0,C 180,E1 1041.022,E2 1041.022} C_VEL
LIN {X 0,Y 601.567,Z 462.44,A -85,B 0,C 180,E1 1046.161,E2 1046.161} C_VEL
LIN {X 0,Y 601.666,Z 462.44,A -85,B 0,C 180,E1 1051.438,E2 1051.438} C_VEL
LIN {X 0,Y 601.726,Z 462.44,A -85,B 0,C 180,E1 1056.261,E2 1056.261} C_VEL
LIN {X 0,Y 601.94,Z 462.44,A -85,B 0,C 180,E1 1060.914,E2 1060.914} C_VEL
LIN {X 0,Y 601.539,Z 462.44,A -85,B 0,C 180,E1 1065.422,E2 1065.422} C_VEL
LIN {X 0,Y 601.986,Z 462.44,A -85,B 0,C 180,E1 1069.86,E2 1069.86} C_VEL
LIN {X 0,Y 602.194,Z 462.44,A -85,B 0,C 180,E1 1074.228,E2 1074.228} C_VEL
LIN {X 0,Y 601.884,Z 462.44,A -85,B 0,C 180,E1 1079.999,E2 1079.999} C_VEL
LIN {X 0,Y 601.918,Z 462.44,A -85,B 0,C 180,E1 1084.327,E2 1084.327} C_VEL
LIN {X 0,Y 601.997,Z 462.44,A -85,B 0,C 180,E1 1088.678,E2 1088.678} C_VEL
LIN {X 0,Y 602.071,Z 462.44,A -85,B 0,C 180,E1 1093.079,E2 1093.079} C_VEL
LIN {X 0,Y 601.806,Z 462.44,A -85,B 0,C 180,E1 1099.088,E2 1099.088} C_VEL
LIN {X 0,Y 601.744,Z 462.44,A -85,B 0,C 180,E1 1103.737,E2 1103.737} C_VEL
LIN {X 0,Y 601.771,Z 462.44,A -85,B 0,C 180,E1 1108.554,E2 1108.554} C_VEL
LIN {X 0,Y 601.904,Z 462.44,A -85,B 0,C 180,E1 1113.887,E2 1113.887} C_VEL
LIN {X 0,Y 601.704,Z 462.44,A -85,B 0,C 180,E1 1118.977,E2 1118.977} C_VEL
LIN {X 0,Y 601.578,Z 462.44,A -85,B 0,C 180,E1 1123.121,E2 1123.121} C_VEL
LIN {X 0,Y 601.7,Z 462.44,A -85,B 0,C 180,E1 1129.136,E2 1129.136} C_VEL
LIN {X 0,Y 601.928,Z 462.44,A -85,B 0,C 180,E1 1134.651,E2 1134.651} C_VEL
LIN {X 0,Y 602.099,Z 462.545,A -85,B 0,C 180,E1 1140.143,E2 1140.143} C_VEL
LIN {X 0,Y 603.295,Z 473.696,A -85,B 0,C 180,E1 1140.358,E2 1140.358} C_VEL
LIN {X 0,Y 603.82,Z 530.696,A -85,B 0,C 180,E1 1141.286,E2 1141.286} C_VEL
LIN {X 0,Y 603.592,Z 570.794,A -85,B 0,C 180,E1 1142.541,E2 1142.541} C_VEL
LIN {X 0,Y 603.3,Z 608.579,A -85,B 0,C 180,E1 1144.347,E2 1144.347} C_VEL
LIN {X 0,Y 602.974,Z 644.394,A -85,B 0,C 180,E1 1146.719,E2 1146.719} C_VEL
LIN {X 0,Y 602.636,Z 676.232,A -85,B 0,C 180,E1 1149.511,E2 1149.511} C_VEL
LIN {X 0,Y 602.417,Z 703.731,A -85,B 0,C 180,E1 1152.658,E2 1152.658} C_VEL
LIN {X 0,Y 602.293,Z 727.014,A -85,B 0,C 180,E1 1156.183,E2 1156.183} C_VEL
LIN {X 0,Y 602.244,Z 744.586,A -85,B 0,C 180,E1 1159.864,E2 1159.864} C_VEL
LIN {X 0,Y 602.229,Z 756.696,A -85,B 0,C 180,E1 1163.726,E2 1163.726} C_VEL
LIN {X 0,Y 602.087,Z 762.448,A -85,B 0,C 180,E1 1167.117,E2 1167.117} C_VEL
LIN {X 0,Y 602.063,Z 763.996,A -85,B 0,C 180,E1 1170,E2 1170} C_VEL
LIN {X 0,Y 602.062,Z 762.341,A -85,B 0,C 180,E1 1172.883,E2 1172.883} C_VEL
LIN {X 0,Y 602.104,Z 756.579,A -85,B 0,C 180,E1 1176.239,E2 1176.239} C_VEL
LIN {X 0,Y 602.089,Z 745.607,A -85,B 0,C 180,E1 1179.773,E2 1179.773} C_VEL
LIN {X 0,Y 602.192,Z 730.512,A -85,B 0,C 180,E1 1183.079,E2 1183.079} C_VEL
LIN {X 0,Y 602.318,Z 710.331,A -85,B 0,C 180,E1 1186.352,E2 1186.352} C_VEL
LIN {X 0,Y 602.529,Z 685.224,A -85,B 0,C 180,E1 1189.46,E2 1189.46} C_VEL
LIN {X 0,Y 602.855,Z 655.41,A -85,B 0,C 180,E1 1192.308,E2 1192.308} C_VEL
LIN {X 0,Y 603.16,Z 621.841,A -85,B 0,C 180,E1 1194.766,E2 1194.766} C_VEL
LIN {X 0,Y 603.498,Z 585.349,A -85,B 0,C 180,E1 1196.746,E2 1196.746} C_VEL
LIN {X 0,Y 603.742,Z 548.119,A -85,B 0,C 180,E1 1198.151,E2 1198.151} C_VEL
LIN {X 0,Y 603.832,Z 511.481,A -85,B 0,C 180,E1 1198.999,E2 1198.999} C_VEL
LIN {X 0,Y 602.998,Z 468.036,A -85,B 0,C 180,E1 1199.644,E2 1199.644} C_VEL
LIN {X 0,Y 602.168,Z 462.44,A -85,B 0,C 180,E1 1199.831,E2 1199.831} C_VEL
LIN {X 0,Y 601.883,Z 462.44,A -85,B 0,C 180,E1 1207.14,E2 1207.14} C_VEL
LIN {X 0,Y 601.566,Z 462.44,A -85,B 0,C 180,E1 1213.128,E2 1213.128} C_VEL
LIN {X 0,Y 601.723,Z 462.44,A -85,B 0,C 180,E1 1219.017,E2 1219.017} C_VEL
LIN {X 0,Y 601.699,Z 462.44,A -85,B 0,C 180,E1 1224.641,E2 1224.641} C_VEL
LIN {X 0,Y 601.811,Z 462.44,A -85,B 0,C 180,E1 1229.794,E2 1229.794} C_VEL
LIN {X 0,Y 602.018,Z 462.44,A -85,B 0,C 180,E1 1234.882,E2 1234.882} C_VEL
LIN {X 0,Y 601.951,Z 462.44,A -85,B 0,C 180,E1 1240.917,E2 1240.917} C_VEL
LIN {X 0,Y 602.15,Z 462.44,A -85,B 0,C 180,E1 1246.923,E2 1246.923} C_VEL
LIN {X 0,Y 601.878,Z 462.44,A -85,B 0,C 180,E1 1252.776,E2 1252.776} C_VEL
LIN {X 0,Y 601.872,Z 462.44,A -85,B 0,C 180,E1 1257.65,E2 1257.65} C_VEL
LIN {X 0,Y 597.828,Z 462.44,A -85,B 0,C 180,E1 1259.275,E2 1259.275} C_VEL
LIN {X 0,Y 594.119,Z 462.44,A -85,B 0,C 180,E1 1260.921,E2 1260.921} C_VEL
LIN {X 0,Y 594.123,Z 462.44,A -85,B 0,C 180,E1 1266.319,E2 1266.319} C_VEL
LIN {X 0,Y 593.922,Z 462.44,A -85,B 0,C 180,E1 1271.767,E2 1271.767} C_VEL
LIN {X 0,Y 593.908,Z 462.44,A -85,B 0,C 180,E1 1276.285,E2 1276.285} C_VEL
LIN {X 0,Y 593.966,Z 462.44,A -85,B 0,C 180,E1 1280.907,E2 1280.907} C_VEL
LIN {X 0,Y 593.97,Z 462.44,A -85,B 0,C 180,E1 1285.679,E2 1285.679} C_VEL
LIN {X 0,Y 593.871,Z 462.44,A -85,B 0,C 180,E1 1290.655,E2 1290.655} C_VEL
LIN {X 0,Y 593.864,Z 462.44,A -85,B 0,C 180,E1 1295.899,E2 1295.899} C_VEL
LIN {X 0,Y 593.799,Z 462.44,A -85,B 0,C 180,E1 1301.522,E2 1301.522} C_VEL
LIN {X 0,Y 593.701,Z 462.44,A -85,B 0,C 180,E1 1306.481,E2 1306.481} C_VEL
LIN {X 0,Y 593.717,Z 462.44,A -85,B 0,C 180,E1 1312.261,E2 1312.261} C_VEL
LIN {X 0,Y 593.896,Z 462.615,A -85,B 0,C 180,E1 1315.42,E2 1315.42} C_VEL
LIN {X 0,Y 597.614,Z 473.546,A -85,B 0,C 180,E1 1315.821,E2 1315.821} C_VEL
LIN {X 0,Y 597.543,Z 529.646,A -85,B 0,C 180,E1 1316.769,E2 1316.769} C_VEL
LIN {X 0,Y 597.162,Z 570.168,A -85,B 0,C 180,E1 1318.056,E2 1318.056} C_VEL
LIN {X 0,Y 596.592,Z 608.626,A -85,B 0,C 180,E1 1319.85,E2 1319.85} C_VEL
LIN {X 0,Y 596.016,Z 646.078,A -85,B 0,C 180,E1 1322.216,E2 1322.216} C_VEL
LIN {X 0,Y 595.381,Z 680.873,A -85,B 0,C 180,E1 1325.074,E2 1325.074} C_VEL
LIN {X 0,Y 594.944,Z 711.011,A -85,B 0,C 180,E1 1328.23,E2 1328.23} C_VEL
LIN {X 0,Y 594.518,Z 737.923,A -85,B 0,C 180,E1 1331.821,E2 1331.821} C_VEL
LIN {X 0,Y 594.318,Z 758.966,A -85,B 0,C 180,E1 1335.47,E2 1335.47} C_VEL
LIN {X 0,Y 594.178,Z 774.964,A -85,B 0,C 180,E1 1339.225,E2 1339.225} C_VEL
LIN {X 0,Y 594.135,Z 785.331,A -85,B 0,C 180,E1 1342.679,E2 1342.679} C_VEL
LIN {X 0,Y 594.284,Z 790.904,A -85,B 0,C 180,E1 1345.616,E2 1345.616} C_VEL
LIN {X 0,Y 594.313,Z 793.657,A -85,B 0,C 180,E1 1348.54,E2 1348.54} C_VEL
LIN {X 0,Y 594.198,Z 792.627,A -85,B 0,C 180,E1 1352.921,E2 1352.921} C_VEL
LIN {X 0,Y 594.311,Z 787.018,A -85,B 0,C 180,E1 1356.535,E2 1356.535} C_VEL
LIN {X 0,Y 594.348,Z 776.777,A -85,B 0,C 180,E1 1360.272,E2 1360.272} C_VEL
LIN {X 0,Y 594.456,Z 760.38,A -85,B 0,C 180,E1 1364.238,E2 1364.238} C_VEL
LIN {X 0,Y 594.66,Z 737.923,A -85,B 0,C 180,E1 1368.174,E2 1368.174} C_VEL
LIN {X 0,Y 595.033,Z 709.61,A -85,B 0,C 180,E1 1371.937,E2 1371.937} C_VEL
LIN {X 0,Y 595.508,Z 676.828,A -85,B 0,C 180,E1 1375.298,E2 1375.298} C_VEL
LIN {X 0,Y 596.123,Z 640.123,A -85,B 0,C 180,E1 1378.208,E2 1378.208} C_VEL
LIN {X 0,Y 596.733,Z 600.78,A -85,B 0,C 180,E1 1380.569,E2 1380.569} C_VEL
LIN {X 0,Y 597.35,Z 560.214,A -85,B 0,C 180,E1 1382.316,E2 1382.316} C_VEL
LIN {X 0,Y 597.676,Z 520.747,A -85,B 0,C 180,E1 1383.42,E2 1383.42} C_VEL
LIN {X 0,Y 597.169,Z 470.335,A -85,B 0,C 180,E1 1384.254,E2 1384.254} C_VEL
LIN {X 0,Y 593.89,Z 462.44,A -85,B 0,C 180,E1 1384.632,E2 1384.632} C_VEL
LIN {X 0,Y 593.691,Z 462.44,A -85,B 0,C 180,E1 1390.09,E2 1390.09} C_VEL
LIN {X 0,Y 593.798,Z 462.44,A -85,B 0,C 180,E1 1395.559,E2 1395.559} C_VEL
LIN {X 0,Y 593.748,Z 462.44,A -85,B 0,C 180,E1 1400.397,E2 1400.397} C_VEL
LIN {X 0,Y 593.679,Z 462.44,A -85,B 0,C 180,E1 1405.872,E2 1405.872} C_VEL
LIN {X 0,Y 593.756,Z 462.44,A -85,B 0,C 180,E1 1411.022,E2 1411.022} C_VEL
LIN {X 0,Y 593.897,Z 462.44,A -85,B 0,C 180,E1 1415.928,E2 1415.928} C_VEL
LIN {X 0,Y 594.026,Z 462.44,A -85,B 0,C 180,E1 1420.65,E2 1420.65} C_VEL
LIN {X 0,Y 593.699,Z 462.44,A -85,B 0,C 180,E1 1425.225,E2 1425.225} C_VEL
LIN {X 0,Y 594.046,Z 462.44,A -85,B 0,C 180,E1 1429.723,E2 1429.723} C_VEL
LIN {X 0,Y 594.257,Z 462.44,A -85,B 0,C 180,E1 1434.15,E2 1434.15} C_VEL
LIN {X 0,Y 593.984,Z 462.44,A -85,B 0,C 180,E1 1439.999,E2 1439.999} C_VEL
LIN {X 0,Y 594.003,Z 462.44,A -85,B 0,C 180,E1 1444.384,E2 1444.384} C_VEL
LIN {X 0,Y 594.079,Z 462.44,A -85,B 0,C 180,E1 1448.794,E2 1448.794} C_VEL
LIN {X 0,Y 593.818,Z 462.44,A -85,B 0,C 180,E1 1454.319,E2 1454.319} C_VEL
LIN {X 0,Y 593.856,Z 462.44,A -85,B 0,C 180,E1 1459.373,E2 1459.373} C_VEL
LIN {X 0,Y 593.805,Z 462.44,A -85,B 0,C 180,E1 1464.074,E2 1464.074} C_VEL
LIN {X 0,Y 593.775,Z 462.44,A -85,B 0,C 180,E1 1468.975,E2 1468.975} C_VEL
LIN {X 0,Y 593.98,Z 462.44,A -85,B 0,C 180,E1 1474.106,E2 1474.106} C_VEL
LIN {X 0,Y 593.729,Z 462.44,A -85,B 0,C 180,E1 1480.087,E2 1480.087} C_VEL
LIN {X 0,Y 593.517,Z 462.44,A -85,B 0,C 180,E1 1485.579,E2 1485.579} C_VEL
LIN {X 0,Y 593.745,Z 462.44,A -85,B 0,C 180,E1 1490.392,E2 1490.392} C_VEL
LIN {X 0,Y 594.085,Z 462.44,A -85,B 0,C 180,E1 1495.895,E2 1495.895} C_VEL
LIN {X 0,Y 594.115,Z 463.048,A -85,B 0,C 180,E1 1499.708,E2 1499.708} C_VEL
LIN {X 0,Y 596.388,Z 470.228,A -85,B 0,C 180,E1 1499.933,E2 1499.933} C_VEL
LIN {X 0,Y 596.864,Z 531.118,A -85,B 0,C 180,E1 1500.931,E2 1500.931} C_VEL
LIN {X 0,Y 596.492,Z 571.538,A -85,B 0,C 180,E1 1502.218,E2 1502.218} C_VEL
LIN {X 0,Y 596.022,Z 609.719,A -85,B 0,C 180,E1 1504.079,E2 1504.079} C_VEL
LIN {X 0,Y 595.493,Z 644.3,A -85,B 0,C 180,E1 1506.402,E2 1506.402} C_VEL
LIN {X 0,Y 595.008,Z 675.169,A -85,B 0,C 180,E1 1509.129,E2 1509.129} C_VEL
LIN {X 0,Y 594.675,Z 702.069,A -85,B 0,C 180,E1 1512.209,E2 1512.209} C_VEL
LIN {X 0,Y 594.415,Z 723.704,A -85,B 0,C 180,E1 1515.427,E2 1515.427} C_VEL
LIN {X 0,Y 594.297,Z 741.334,A -85,B 0,C 180,E1 1518.942,E2 1518.942} C_VEL
LIN {X 0,Y 594.227,Z 754.23,A -85,B 0,C 180,E1 1522.68,E2 1522.68} C_VEL
LIN {X 0,Y 594.137,Z 760.506,A -85,B 0,C 180,E1 1525.615,E2 1525.615} C_VEL
LIN {X 0,Y 594.149,Z 763.614,A -85,B 0,C 180,E1 1528.54,E2 1528.54} C_VEL
LIN {X 0,Y 594.293,Z 763.551,A -85,B 0,C 180,E1 1531.46,E2 1531.46} C_VEL
LIN {X 0,Y 594.352,Z 759.139,A -85,B 0,C 180,E1 1535.116,E2 1535.116} C_VEL
LIN {X 0,Y 594.318,Z 749.568,A -85,B 0,C 180,E1 1538.793,E2 1538.793} C_VEL
LIN {X 0,Y 594.38,Z 734.365,A -85,B 0,C 180,E1 1542.505,E2 1542.505} C_VEL
LIN {X 0,Y 594.555,Z 712.466,A -85,B 0,C 180,E1 1546.268,E2 1546.268} C_VEL
LIN {X 0,Y 594.84,Z 687.008,A -85,B 0,C 180,E1 1549.526,E2 1549.526} C_VEL
LIN {X 0,Y 595.308,Z 657.491,A -85,B 0,C 180,E1 1552.428,E2 1552.428} C_VEL
LIN {X 0,Y 595.8,Z 624.091,A -85,B 0,C 180,E1 1554.945,E2 1554.945} C_VEL
LIN {X 0,Y 596.318,Z 588.54,A -85,B 0,C 180,E1 1556.941,E2 1556.941} C_VEL
LIN {X 0,Y 596.674,Z 551.231,A -85,B 0,C 180,E1 1558.417,E2 1558.417} C_VEL
LIN {X 0,Y 596.915,Z 512.112,A -85,B 0,C 180,E1 1559.359,E2 1559.359} C_VEL
LIN {X 0,Y 596.014,Z 467.91,A -85,B 0,C 180,E1 1560.029,E2 1560.029} C_VEL
LIN {X 0,Y 594.101,Z 462.44,A -85,B 0,C 180,E1 1560.286,E2 1560.286} C_VEL
LIN {X 0,Y 593.89,Z 462.44,A -85,B 0,C 180,E1 1565.901,E2 1565.901} C_VEL
LIN {X 0,Y 593.6,Z 462.44,A -85,B 0,C 180,E1 1571.544,E2 1571.544} C_VEL
LIN {X 0,Y 593.769,Z 462.44,A -85,B 0,C 180,E1 1576.495,E2 1576.495} C_VEL
LIN {X 0,Y 593.754,Z 462.44,A -85,B 0,C 180,E1 1582.27,E2 1582.27} C_VEL
LIN {X 0,Y 593.636,Z 462.44,A -85,B 0,C 180,E1 1587.619,E2 1587.619} C_VEL
LIN {X 0,Y 593.719,Z 462.44,A -85,B 0,C 180,E1 1592.679,E2 1592.679} C_VEL
LIN {X 0,Y 593.712,Z 462.44,A -85,B 0,C 180,E1 1597.512,E2 1597.512} C_VEL
LIN {X 0,Y 593.964,Z 462.44,A -85,B 0,C 180,E1 1602.191,E2 1602.191} C_VEL
LIN {X 0,Y 594.208,Z 462.44,A -85,B 0,C 180,E1 1606.745,E2 1606.745} C_VEL
LIN {X 0,Y 593.994,Z 462.44,A -85,B 0,C 180,E1 1612.679,E2 1612.679} C_VEL
LIN {X 0,Y 593.965,Z 462.44,A -85,B 0,C 180,E1 1617.636,E2 1617.636} C_VEL
LIN {X 0,Y 594.119,Z 462.44,A -85,B 0,C 180,E1 1620.921,E2 1620.921} C_VEL
LIN {X 0,Y 591.615,Z 462.44,A -85,B 0,C 180,E1 1622.165,E2 1622.165} C_VEL
LIN {X 0,Y 586.101,Z 462.44,A -85,B 0,C 180,E1 1624.025,E2 1624.025} C_VEL
LIN {X 0,Y 586.024,Z 462.44,A -85,B 0,C 180,E1 1624.24,E2 1624.24} C_VEL
LIN {X 0,Y 585.947,Z 462.44,A -85,B 0,C 180,E1 1628.919,E2 1628.919} C_VEL
LIN {X 0,Y 585.967,Z 462.44,A -85,B 0,C 180,E1 1633.447,E2 1633.447} C_VEL
LIN {X 0,Y 585.869,Z 462.44,A -85,B 0,C 180,E1 1638.066,E2 1638.066} C_VEL
LIN {X 0,Y 585.872,Z 462.44,A -85,B 0,C 180,E1 1642.807,E2 1642.807} C_VEL
LIN {X 0,Y 585.801,Z 462.44,A -85,B 0,C 180,E1 1647.724,E2 1647.724} C_VEL
LIN {X 0,Y 585.736,Z 462.44,A -85,B 0,C 180,E1 1652.875,E2 1652.875} C_VEL
LIN {X 0,Y 585.852,Z 462.44,A -85,B 0,C 180,E1 1658.332,E2 1658.332} C_VEL
LIN {X 0,Y 585.91,Z 462.44,A -85,B 0,C 180,E1 1664.241,E2 1664.241} C_VEL
LIN {X 0,Y 585.795,Z 462.44,A -85,B 0,C 180,E1 1669.745,E2 1669.745} C_VEL
LIN {X 0,Y 585.859,Z 462.658,A -85,B 0,C 180,E1 1674.877,E2 1674.877} C_VEL
LIN {X 0,Y 591.001,Z 473.782,A -85,B 0,C 180,E1 1675.388,E2 1675.388} C_VEL
LIN {X 0,Y 590.903,Z 529.891,A -85,B 0,C 180,E1 1676.352,E2 1676.352} C_VEL
LIN {X 0,Y 590.353,Z 570.849,A -85,B 0,C 180,E1 1677.67,E2 1677.67} C_VEL
LIN {X 0,Y 589.602,Z 608.629,A -85,B 0,C 180,E1 1679.455,E2 1679.455} C_VEL
LIN {X 0,Y 588.78,Z 646.214,A -85,B 0,C 180,E1 1681.854,E2 1681.854} C_VEL
LIN {X 0,Y 587.956,Z 680.827,A -85,B 0,C 180,E1 1684.732,E2 1684.732} C_VEL
LIN {X 0,Y 587.289,Z 711.73,A -85,B 0,C 180,E1 1688.02,E2 1688.02} C_VEL
LIN {X 0,Y 586.756,Z 737.924,A -85,B 0,C 180,E1 1691.572,E2 1691.572} C_VEL
LIN {X 0,Y 586.482,Z 759.634,A -85,B 0,C 180,E1 1695.404,E2 1695.404} C_VEL
LIN {X 0,Y 586.322,Z 775.536,A -85,B 0,C 180,E1 1699.238,E2 1699.238} C_VEL
LIN {X 0,Y 586.245,Z 785.33,A -85,B 0,C 180,E1 1702.58,E2 1702.58} C_VEL
LIN {X 0,Y 586.388,Z 790.904,A -85,B 0,C 180,E1 1705.557,E2 1705.557} C_VEL
LIN {X 0,Y 586.408,Z 793.657,A -85,B 0,C 180,E1 1708.52,E2 1708.52} C_VEL
LIN {X 0,Y 586.298,Z 792.627,A -85,B 0,C 180,E1 1712.961,E2 1712.961} C_VEL
LIN {X 0,Y 586.405,Z 787.018,A -85,B 0,C 180,E1 1716.624,E2 1716.624} C_VEL
LIN {X 0,Y 586.443,Z 776.777,A -85,B 0,C 180,E1 1720.412,E2 1720.412} C_VEL
LIN {X 0,Y 586.587,Z 759.369,A -85,B 0,C 180,E1 1724.646,E2 1724.646} C_VEL
LIN {X 0,Y 586.856,Z 736.696,A -85,B 0,C 180,E1 1728.62,E2 1728.62} C_VEL
LIN {X 0,Y 587.397,Z 708.491,A -85,B 0,C 180,E1 1732.368,E2 1732.368} C_VEL
LIN {X 0,Y 588.058,Z 676.193,A -85,B 0,C 180,E1 1735.699,E2 1735.699} C_VEL
LIN {X 0,Y 588.919,Z 639.662,A -85,B 0,C 180,E1 1738.616,E2 1738.616} C_VEL
LIN {X 0,Y 589.788,Z 600.658,A -85,B 0,C 180,E1 1740.975,E2 1740.975} C_VEL
LIN {X 0,Y 590.584,Z 560.212,A -85,B 0,C 180,E1 1742.732,E2 1742.732} C_VEL
LIN {X 0,Y 591.046,Z 521.632,A -85,B 0,C 180,E1 1743.825,E2 1743.825} C_VEL
LIN {X 0,Y 590.423,Z 472.521,A -85,B 0,C 180,E1 1744.669,E2 1744.669} C_VEL
LIN {X 0,Y 585.857,Z 462.44,A -85,B 0,C 180,E1 1745.176,E2 1745.176} C_VEL
LIN {X 0,Y 585.796,Z 462.44,A -85,B 0,C 180,E1 1750.255,E2 1750.255} C_VEL
LIN {X 0,Y 585.929,Z 462.44,A -85,B 0,C 180,E1 1756.35,E2 1756.35} C_VEL
LIN {X 0,Y 585.852,Z 462.44,A -85,B 0,C 180,E1 1761.668,E2 1761.668} C_VEL
LIN {X 0,Y 585.744,Z 462.44,A -85,B 0,C 180,E1 1767.126,E2 1767.126} C_VEL
LIN {X 0,Y 585.799,Z 462.44,A -85,B 0,C 180,E1 1772.276,E2 1772.276} C_VEL
LIN {X 0,Y 585.861,Z 462.44,A -85,B 0,C 180,E1 1777.192,E2 1777.192} C_VEL
LIN {X 0,Y 586.095,Z 462.44,A -85,B 0,C 180,E1 1781.941,E2 1781.941} C_VEL
LIN {X 0,Y 585.816,Z 462.44,A -85,B 0,C 180,E1 1788.067,E2 1788.067} C_VEL
LIN {X 0,Y 586.336,Z 462.44,A -85,B 0,C 180,E1 1794.071,E2 1794.071} C_VEL
LIN {X 0,Y 586.094,Z 462.44,A -85,B 0,C 180,E1 1799.999,E2 1799.999} C_VEL
LIN {X 0,Y 586.099,Z 462.44,A -85,B 0,C 180,E1 1804.444,E2 1804.444} C_VEL
LIN {X 0,Y 586.142,Z 462.44,A -85,B 0,C 180,E1 1808.914,E2 1808.914} C_VEL
LIN {X 0,Y 586.149,Z 462.44,A -85,B 0,C 180,E1 1813.441,E2 1813.441} C_VEL
LIN {X 0,Y 586.066,Z 462.44,A -85,B 0,C 180,E1 1818.058,E2 1818.058} C_VEL
LIN {X 0,Y 585.997,Z 462.44,A -85,B 0,C 180,E1 1822.8,E2 1822.8} C_VEL
LIN {X 0,Y 585.843,Z 462.44,A -85,B 0,C 180,E1 1828.509,E2 1828.509} C_VEL
LIN {X 0,Y 586.021,Z 462.44,A -85,B 0,C 180,E1 1834.635,E2 1834.635} C_VEL
LIN {X 0,Y 585.842,Z 462.44,A -85,B 0,C 180,E1 1840.244,E2 1840.244} C_VEL
LIN {X 0,Y 585.694,Z 462.44,A -85,B 0,C 180,E1 1846.365,E2 1846.365} C_VEL
LIN {X 0,Y 585.876,Z 462.44,A -85,B 0,C 180,E1 1851.665,E2 1851.665} C_VEL
LIN {X 0,Y 586.127,Z 462.44,A -85,B 0,C 180,E1 1857.147,E2 1857.147} C_VEL
LIN {X 0,Y 586.149,Z 462.44,A -85,B 0,C 180,E1 1859.224,E2 1859.224} C_VEL
LIN {X 0,Y 589.574,Z 473.507,A -85,B 0,C 180,E1 1859.595,E2 1859.595} C_VEL
LIN {X 0,Y 589.932,Z 531.25,A -85,B 0,C 180,E1 1860.56,E2 1860.56} C_VEL
LIN {X 0,Y 589.453,Z 571.018,A -85,B 0,C 180,E1 1861.836,E2 1861.836} C_VEL
LIN {X 0,Y 588.779,Z 609.07,A -85,B 0,C 180,E1 1863.698,E2 1863.698} C_VEL
LIN {X 0,Y 588.047,Z 644.294,A -85,B 0,C 180,E1 1866.085,E2 1866.085} C_VEL
LIN {X 0,Y 587.425,Z 675.163,A -85,B 0,C 180,E1 1868.847,E2 1868.847} C_VEL
LIN {X 0,Y 586.937,Z 702.065,A -85,B 0,C 180,E1 1871.967,E2 1871.967} C_VEL
LIN {X 0,Y 586.592,Z 724.416,A -85,B 0,C 180,E1 1875.353,E2 1875.353} C_VEL
LIN {X 0,Y 586.424,Z 741.442,A -85,B 0,C 180,E1 1878.818,E2 1878.818} C_VEL
LIN {X 0,Y 586.33,Z 754.229,A -85,B 0,C 180,E1 1882.581,E2 1882.581} C_VEL
LIN {X 0,Y 586.238,Z 760.505,A -85,B 0,C 180,E1 1885.556,E2 1885.556} C_VEL
LIN {X 0,Y 586.256,Z 763.614,A -85,B 0,C 180,E1 1888.52,E2 1888.52} C_VEL
LIN {X 0,Y 586.388,Z 763.552,A -85,B 0,C 180,E1 1891.48,E2 1891.48} C_VEL
LIN {X 0,Y 586.452,Z 759.14,A -85,B 0,C 180,E1 1895.185,E2 1895.185} C_VEL
LIN {X 0,Y 586.413,Z 749.57,A -85,B 0,C 180,E1 1898.912,E2 1898.912} C_VEL
LIN {X 0,Y 586.517,Z 734.369,A -85,B 0,C 180,E1 1902.676,E2 1902.676} C_VEL
LIN {X 0,Y 586.758,Z 713.772,A -85,B 0,C 180,E1 1906.298,E2 1906.298} C_VEL
LIN {X 0,Y 587.206,Z 687.264,A -85,B 0,C 180,E1 1909.762,E2 1909.762} C_VEL
LIN {X 0,Y 587.763,Z 657.5,A -85,B 0,C 180,E1 1912.732,E2 1912.732} C_VEL
LIN {X 0,Y 588.466,Z 624.129,A -85,B 0,C 180,E1 1915.276,E2 1915.276} C_VEL
LIN {X 0,Y 589.158,Z 589.333,A -85,B 0,C 180,E1 1917.258,E2 1917.258} C_VEL
LIN {X 0,Y 589.685,Z 552.414,A -85,B 0,C 180,E1 1918.748,E2 1918.748} C_VEL
LIN {X 0,Y 590.019,Z 513.803,A -85,B 0,C 180,E1 1919.709,E2 1919.709} C_VEL
LIN {X 0,Y 589.312,Z 470.797,A -85,B 0,C 180,E1 1920.367,E2 1920.367} C_VEL
LIN {X 0,Y 586.088,Z 462.44,A -85,B 0,C 180,E1 1920.735,E2 1920.735} C_VEL
LIN {X 0,Y 585.957,Z 462.44,A -85,B 0,C 180,E1 1926.78,E2 1926.78} C_VEL
LIN {X 0,Y 585.698,Z 462.44,A -85,B 0,C 180,E1 1932.233,E2 1932.233} C_VEL
LIN {X 0,Y 585.876,Z 462.44,A -85,B 0,C 180,E1 1937.79,E2 1937.79} C_VEL
LIN {X 0,Y 585.824,Z 462.44,A -85,B 0,C 180,E1 1943.532,E2 1943.532} C_VEL
LIN {X 0,Y 585.853,Z 462.44,A -85,B 0,C 180,E1 1948.881,E2 1948.881} C_VEL
LIN {X 0,Y 585.998,Z 462.44,A -85,B 0,C 180,E1 1954.736,E2 1954.736} C_VEL
LIN {X 0,Y 586.129,Z 462.44,A -85,B 0,C 180,E1 1960.381,E2 1960.381} C_VEL
LIN {X 0,Y 586.283,Z 462.44,A -85,B 0,C 180,E1 1966.562,E2 1966.562} C_VEL
LIN {X 0,Y 586.091,Z 462.44,A -85,B 0,C 180,E1 1972.58,E2 1972.58} C_VEL
LIN {X 0,Y 586.213,Z 462.44,A -85,B 0,C 180,E1 1977.04,E2 1977.04} C_VEL
LIN {X 0,Y 586.353,Z 462.44,A -85,B 0,C 180,E1 1981.48,E2 1981.48} C_VEL
LIN {X 0,Y 586.024,Z 462.44,A -85,B 0,C 180,E1 1984.24,E2 1984.24} C_VEL
LIN {X 0,Y 583.597,Z 462.44,A -85,B 0,C 180,E1 1985.503,E2 1985.503} C_VEL
LIN {X 0,Y 578.083,Z 462.44,A -85,B 0,C 180,E1 1987.612,E2 1987.612} C_VEL
LIN {X 0,Y 578.094,Z 462.44,A -85,B 0,C 180,E1 1992.094,E2 1992.094} C_VEL
LIN {X 0,Y 578.046,Z 462.44,A -85,B 0,C 180,E1 1996.745,E2 1996.745} C_VEL
LIN {X 0,Y 578.059,Z 462.44,A -85,B 0,C 180,E1 2001.511,E2 2001.511} C_VEL
LIN {X 0,Y 577.946,Z 462.44,A -85,B 0,C 180,E1 2007.032,E2 2007.032} C_VEL
LIN {X 0,Y 577.911,Z 462.44,A -85,B 0,C 180,E1 2011.598,E2 2011.598} C_VEL
LIN {X 0,Y 577.97,Z 462.44,A -85,B 0,C 180,E1 2017.048,E2 2017.048} C_VEL
LIN {X 0,Y 577.975,Z 462.44,A -85,B 0,C 180,E1 2022.927,E2 2022.927} C_VEL
LIN {X 0,Y 577.834,Z 462.44,A -85,B 0,C 180,E1 2029.073,E2 2029.073} C_VEL
LIN {X 0,Y 577.871,Z 462.44,A -85,B 0,C 180,E1 2034.309,E2 2034.309} C_VEL
LIN {X 0,Y 584.583,Z 478.755,A -85,B 0,C 180,E1 2035.025,E2 2035.025} C_VEL
LIN {X 0,Y 584.33,Z 529.641,A -85,B 0,C 180,E1 2035.916,E2 2035.916} C_VEL
LIN {X 0,Y 583.583,Z 569.503,A -85,B 0,C 180,E1 2037.194,E2 2037.194} C_VEL
LIN {X 0,Y 582.752,Z 606.113,A -85,B 0,C 180,E1 2038.911,E2 2038.911} C_VEL
LIN {X 0,Y 581.667,Z 643.996,A -85,B 0,C 180,E1 2041.309,E2 2041.309} C_VEL
LIN {X 0,Y 580.535,Z 679.748,A -85,B 0,C 180,E1 2044.28,E2 2044.28} C_VEL
LIN {X 0,Y 579.663,Z 710.871,A -85,B 0,C 180,E1 2047.608,E2 2047.608} C_VEL
LIN {X 0,Y 578.993,Z 738.041,A -85,B 0,C 180,E1 2051.334,E2 2051.334} C_VEL
LIN {X 0,Y 578.659,Z 759.756,A -85,B 0,C 180,E1 2055.228,E2 2055.228} C_VEL
LIN {X 0,Y 578.437,Z 775.537,A -85,B 0,C 180,E1 2059.09,E2 2059.09} C_VEL
LIN {X 0,Y 578.375,Z 785.33,A -85,B 0,C 180,E1 2062.479,E2 2062.479} C_VEL
LIN {X 0,Y 578.492,Z 790.904,A -85,B 0,C 180,E1 2065.496,E2 2065.496} C_VEL
LIN {X 0,Y 578.503,Z 793.657,A -85,B 0,C 180,E1 2068.5,E2 2068.5} C_VEL
LIN {X 0,Y 578.392,Z 792.627,A -85,B 0,C 180,E1 2073.001,E2 2073.001} C_VEL
LIN {X 0,Y 578.511,Z 786.916,A -85,B 0,C 180,E1 2076.764,E2 2076.764} C_VEL
LIN {X 0,Y 578.549,Z 775.474,A -85,B 0,C 180,E1 2080.926,E2 2080.926} C_VEL
LIN {X 0,Y 578.747,Z 759.611,A -85,B 0,C 180,E1 2084.8,E2 2084.8} C_VEL
LIN {X 0,Y 579.102,Z 736.902,A -85,B 0,C 180,E1 2088.846,E2 2088.846} C_VEL
LIN {X 0,Y 579.808,Z 708.982,A -85,B 0,C 180,E1 2092.62,E2 2092.62} C_VEL
LIN {X 0,Y 580.678,Z 676.194,A -85,B 0,C 180,E1 2096.05,E2 2096.05} C_VEL
LIN {X 0,Y 581.779,Z 640.464,A -85,B 0,C 180,E1 2098.945,E2 2098.945} C_VEL
LIN {X 0,Y 582.872,Z 601.001,A -85,B 0,C 180,E1 2101.367,E2 2101.367} C_VEL
LIN {X 0,Y 583.852,Z 560.951,A -85,B 0,C 180,E1 2103.128,E2 2103.128} C_VEL
LIN {X 0,Y 584.48,Z 521.842,A -85,B 0,C 180,E1 2104.253,E2 2104.253} C_VEL
LIN {X 0,Y 584.134,Z 476.095,A -85,B 0,C 180,E1 2105.044,E2 2105.044} C_VEL
LIN {X 0,Y 577.872,Z 462.44,A -85,B 0,C 180,E1 2105.691,E2 2105.691} C_VEL
LIN {X 0,Y 577.84,Z 462.44,A -85,B 0,C 180,E1 2110.926,E2 2110.926} C_VEL
LIN {X 0,Y 577.978,Z 462.44,A -85,B 0,C 180,E1 2117.074,E2 2117.074} C_VEL
LIN {X 0,Y 577.962,Z 462.44,A -85,B 0,C 180,E1 2122.951,E2 2122.951} C_VEL
LIN {X 0,Y 577.916,Z 462.44,A -85,B 0,C 180,E1 2128.402,E2 2128.402} C_VEL
LIN {X 0,Y 578.006,Z 462.44,A -85,B 0,C 180,E1 2133.558,E2 2133.558} C_VEL
LIN {X 0,Y 578.049,Z 462.44,A -85,B 0,C 180,E1 2138.489,E2 2138.489} C_VEL
LIN {X 0,Y 578.212,Z 462.44,A -85,B 0,C 180,E1 2143.26,E2 2143.26} C_VEL
LIN {X 0,Y 578.173,Z 462.44,A -85,B 0,C 180,E1 2149.437,E2 2149.437} C_VEL
LIN {X 0,Y 578.437,Z 462.44,A -85,B 0,C 180,E1 2154.098,E2 2154.098} C_VEL
LIN {X 0,Y 578.194,Z 462.44,A -85,B 0,C 180,E1 2159.999,E2 2159.999} C_VEL
LIN {X 0,Y 578.186,Z 462.44,A -85,B 0,C 180,E1 2164.505,E2 2164.505} C_VEL
LIN {X 0,Y 578.21,Z 462.44,A -85,B 0,C 180,E1 2169.038,E2 2169.038} C_VEL
LIN {X 0,Y 578.047,Z 462.44,A -85,B 0,C 180,E1 2174.263,E2 2174.263} C_VEL
LIN {X 0,Y 578.031,Z 462.44,A -85,B 0,C 180,E1 2179.906,E2 2179.906} C_VEL
LIN {X 0,Y 577.942,Z 462.44,A -85,B 0,C 180,E1 2184.779,E2 2184.779} C_VEL
LIN {X 0,Y 577.856,Z 462.44,A -85,B 0,C 180,E1 2190.153,E2 2190.153} C_VEL
LIN {X 0,Y 578.012,Z 462.44,A -85,B 0,C 180,E1 2195.185,E2 2195.185} C_VEL
LIN {X 0,Y 577.907,Z 462.44,A -85,B 0,C 180,E1 2200.913,E2 2200.913} C_VEL
LIN {X 0,Y 577.825,Z 462.44,A -85,B 0,C 180,E1 2207.19,E2 2207.19} C_VEL
LIN {X 0,Y 578.039,Z 462.44,A -85,B 0,C 180,E1 2212.953,E2 2212.953} C_VEL
LIN {X 0,Y 578.214,Z 462.44,A -85,B 0,C 180,E1 2218.745,E2 2218.745} C_VEL
LIN {X 0,Y 582.7,Z 473.839,A -85,B 0,C 180,E1 2219.203,E2 2219.203} C_VEL
LIN {X 0,Y 583.023,Z 531.879,A -85,B 0,C 180,E1 2220.194,E2 2220.194} C_VEL
LIN {X 0,Y 582.388,Z 572.074,A -85,B 0,C 180,E1 2221.51,E2 2221.51} C_VEL
LIN {X 0,Y 581.587,Z 608.993,A -85,B 0,C 180,E1 2223.343,E2 2223.343} C_VEL
LIN {X 0,Y 580.673,Z 643.967,A -85,B 0,C 180,E1 2225.735,E2 2225.735} C_VEL
LIN {X 0,Y 579.794,Z 675.156,A -85,B 0,C 180,E1 2228.555,E2 2228.555} C_VEL
LIN {X 0,Y 579.22,Z 702.061,A -85,B 0,C 180,E1 2231.718,E2 2231.718} C_VEL
LIN {X 0,Y 578.779,Z 724.863,A -85,B 0,C 180,E1 2235.231,E2 2235.231} C_VEL
LIN {X 0,Y 578.58,Z 743.016,A -85,B 0,C 180,E1 2239.055,E2 2239.055} C_VEL
LIN {X 0,Y 578.486,Z 755.285,A -85,B 0,C 180,E1 2242.896,E2 2242.896} C_VEL
LIN {X 0,Y 578.34,Z 760.504,A -85,B 0,C 180,E1 2245.495,E2 2245.495} C_VEL
LIN {X 0,Y 578.355,Z 763.613,A -85,B 0,C 180,E1 2248.5,E2 2248.5} C_VEL
LIN {X 0,Y 578.483,Z 763.552,A -85,B 0,C 180,E1 2251.5,E2 2251.5} C_VEL
LIN {X 0,Y 578.557,Z 759.173,A -85,B 0,C 180,E1 2255.239,E2 2255.239} C_VEL
LIN {X 0,Y 578.52,Z 749.572,A -85,B 0,C 180,E1 2259.035,E2 2259.035} C_VEL
LIN {X 0,Y 578.677,Z 734.373,A -85,B 0,C 180,E1 2262.85,E2 2262.85} C_VEL
LIN {X 0,Y 578.976,Z 713.777,A -85,B 0,C 180,E1 2266.523,E2 2266.523} C_VEL
LIN {X 0,Y 579.564,Z 687.276,A -85,B 0,C 180,E1 2270.033,E2 2270.033} C_VEL
LIN {X 0,Y 580.255,Z 657.509,A -85,B 0,C 180,E1 2273.043,E2 2273.043} C_VEL
LIN {X 0,Y 581.169,Z 623.894,A -85,B 0,C 180,E1 2275.633,E2 2275.633} C_VEL
LIN {X 0,Y 582.062,Z 587.855,A -85,B 0,C 180,E1 2277.693,E2 2277.693} C_VEL
LIN {X 0,Y 582.772,Z 550.873,A -85,B 0,C 180,E1 2279.173,E2 2279.173} C_VEL
LIN {X 0,Y 583.174,Z 513.051,A -85,B 0,C 180,E1 2280.107,E2 2280.107} C_VEL
LIN {X 0,Y 582.706,Z 473.739,A -85,B 0,C 180,E1 2280.708,E2 2280.708} C_VEL
LIN {X 0,Y 578.067,Z 462.44,A -85,B 0,C 180,E1 2281.19,E2 2281.19} C_VEL
LIN {X 0,Y 578.043,Z 462.44,A -85,B 0,C 180,E1 2287.047,E2 2287.047} C_VEL
LIN {X 0,Y 577.813,Z 462.44,A -85,B 0,C 180,E1 2292.947,E2 2292.947} C_VEL
LIN {X 0,Y 577.919,Z 462.44,A -85,B 0,C 180,E1 2299.088,E2 2299.088} C_VEL
LIN {X 0,Y 577.845,Z 462.44,A -85,B 0,C 180,E1 2304.803,E2 2304.803} C_VEL
LIN {X 0,Y 577.923,Z 462.44,A -85,B 0,C 180,E1 2310.151,E2 2310.151} C_VEL
LIN {X 0,Y 578.081,Z 462.44,A -85,B 0,C 180,E1 2315.228,E2 2315.228} C_VEL
LIN {X 0,Y 578.205,Z 462.44,A -85,B 0,C 180,E1 2320.515,E2 2320.515} C_VEL
LIN {X 0,Y 578.339,Z 462.44,A -85,B 0,C 180,E1 2326.374,E2 2326.374} C_VEL
LIN {X 0,Y 578.196,Z 462.44,A -85,B 0,C 180,E1 2332.478,E2 2332.478} C_VEL
LIN {X 0,Y 578.306,Z 462.44,A -85,B 0,C 180,E1 2337,E2 2337} C_VEL
LIN {X 0,Y 578.442,Z 462.44,A -85,B 0,C 180,E1 2341.501,E2 2341.501} C_VEL
LIN {X 0,Y 578.4,Z 462.44,A -85,B 0,C 180,E1 2346.011,E2 2346.011} C_VEL
LIN {X 0,Y 578.083,Z 462.44,A -85,B 0,C 180,E1 2347.612,E2 2347.612} C_VEL
LIN {X 0,Y 574.197,Z 462.44,A -85,B 0,C 180,E1 2349.304,E2 2349.304} C_VEL
LIN {X 0,Y 570.265,Z 462.44,A -85,B 0,C 180,E1 2351.018,E2 2351.018} C_VEL
LIN {X 0,Y 570.099,Z 462.44,A -85,B 0,C 180,E1 2357.034,E2 2357.034} C_VEL
LIN {X 0,Y 570.131,Z 462.44,A -85,B 0,C 180,E1 2361.825,E2 2361.825} C_VEL
LIN {X 0,Y 570.075,Z 462.44,A -85,B 0,C 180,E1 2366.839,E2 2366.839} C_VEL
LIN {X 0,Y 569.951,Z 462.44,A -85,B 0,C 180,E1 2372.091,E2 2372.091} C_VEL
LIN {X 0,Y 570.056,Z 462.44,A -85,B 0,C 180,E1 2377.651,E2 2377.651} C_VEL
LIN {X 0,Y 569.984,Z 462.44,A -85,B 0,C 180,E1 2383.678,E2 2383.678} C_VEL
LIN {X 0,Y 569.863,Z 462.44,A -85,B 0,C 180,E1 2388.375,E2 2388.375} C_VEL
LIN {X 0,Y 569.948,Z 463.153,A -85,B 0,C 180,E1 2393.751,E2 2393.751} C_VEL
LIN {X 0,Y 578.118,Z 480.19,A -85,B 0,C 180,E1 2394.597,E2 2394.597} C_VEL
LIN {X 0,Y 577.734,Z 530.82,A -85,B 0,C 180,E1 2395.504,E2 2395.504} C_VEL
LIN {X 0,Y 576.826,Z 572.594,A -85,B 0,C 180,E1 2396.885,E2 2396.885} C_VEL
LIN {X 0,Y 575.628,Z 611.191,A -85,B 0,C 180,E1 2398.78,E2 2398.78} C_VEL
LIN {X 0,Y 574.363,Z 647.493,A -85,B 0,C 180,E1 2401.182,E2 2401.182} C_VEL
LIN {X 0,Y 573.082,Z 681.343,A -85,B 0,C 180,E1 2404.08,E2 2404.08} C_VEL
LIN {X 0,Y 572.021,Z 712.494,A -85,B 0,C 180,E1 2407.498,E2 2407.498} C_VEL
LIN {X 0,Y 571.276,Z 738.238,A -85,B 0,C 180,E1 2411.105,E2 2411.105} C_VEL
LIN {X 0,Y 570.822,Z 759.439,A -85,B 0,C 180,E1 2414.954,E2 2414.954} C_VEL
LIN {X 0,Y 570.565,Z 775.918,A -85,B 0,C 180,E1 2419.047,E2 2419.047} C_VEL
LIN {X 0,Y 570.489,Z 785.33,A -85,B 0,C 180,E1 2422.374,E2 2422.374} C_VEL
LIN {X 0,Y 570.62,Z 790.904,A -85,B 0,C 180,E1 2425.434,E2 2425.434} C_VEL
LIN {X 0,Y 570.603,Z 793.657,A -85,B 0,C 180,E1 2428.479,E2 2428.479} C_VEL
LIN {X 0,Y 570.486,Z 792.627,A -85,B 0,C 180,E1 2433.043,E2 2433.043} C_VEL
LIN {X 0,Y 570.601,Z 786.916,A -85,B 0,C 180,E1 2436.858,E2 2436.858} C_VEL
LIN {X 0,Y 570.652,Z 775.755,A -85,B 0,C 180,E1 2440.999,E2 2440.999} C_VEL
LIN {X 0,Y 570.929,Z 759.311,A -85,B 0,C 180,E1 2445.068,E2 2445.068} C_VEL
LIN {X 0,Y 571.356,Z 736.108,A -85,B 0,C 180,E1 2449.233,E2 2449.233} C_VEL
LIN {X 0,Y 572.226,Z 708.166,A -85,B 0,C 180,E1 2453.032,E2 2453.032} C_VEL
LIN {X 0,Y 573.33,Z 675.361,A -85,B 0,C 180,E1 2456.486,E2 2456.486} C_VEL
LIN {X 0,Y 574.666,Z 639.3,A -85,B 0,C 180,E1 2459.421,E2 2459.421} C_VEL
LIN {X 0,Y 575.989,Z 600.91,A -85,B 0,C 180,E1 2461.79,E2 2461.79} C_VEL
LIN {X 0,Y 577.211,Z 559.843,A -85,B 0,C 180,E1 2463.604,E2 2463.604} C_VEL
LIN {X 0,Y 577.958,Z 522.151,A -85,B 0,C 180,E1 2464.687,E2 2464.687} C_VEL
LIN {X 0,Y 577.679,Z 478.983,A -85,B 0,C 180,E1 2465.452,E2 2465.452} C_VEL
LIN {X 0,Y 569.935,Z 462.44,A -85,B 0,C 180,E1 2466.281,E2 2466.281} C_VEL
LIN {X 0,Y 569.86,Z 462.44,A -85,B 0,C 180,E1 2471.936,E2 2471.936} C_VEL
LIN {X 0,Y 569.986,Z 462.44,A -85,B 0,C 180,E1 2478.056,E2 2478.056} C_VEL
LIN {X 0,Y 569.998,Z 462.44,A -85,B 0,C 180,E1 2484.243,E2 2484.243} C_VEL
LIN {X 0,Y 570.031,Z 462.44,A -85,B 0,C 180,E1 2489.693,E2 2489.693} C_VEL
LIN {X 0,Y 570.135,Z 462.44,A -85,B 0,C 180,E1 2494.857,E2 2494.857} C_VEL
LIN {X 0,Y 570.213,Z 462.44,A -85,B 0,C 180,E1 2499.808,E2 2499.808} C_VEL
LIN {X 0,Y 570.056,Z 462.44,A -85,B 0,C 180,E1 2504.598,E2 2504.598} C_VEL
LIN {X 0,Y 570.16,Z 462.44,A -85,B 0,C 180,E1 2510.832,E2 2510.832} C_VEL
LIN {X 0,Y 570.265,Z 462.44,A -85,B 0,C 180,E1 2515.431,E2 2515.431} C_VEL
LIN {X 0,Y 570.307,Z 462.44,A -85,B 0,C 180,E1 2519.999,E2 2519.999} C_VEL
LIN {X 0,Y 570.289,Z 462.44,A -85,B 0,C 180,E1 2524.567,E2 2524.567} C_VEL
LIN {X 0,Y 570.277,Z 462.44,A -85,B 0,C 180,E1 2529.165,E2 2529.165} C_VEL
LIN {X 0,Y 570.251,Z 462.44,A -85,B 0,C 180,E1 2533.823,E2 2533.823} C_VEL
LIN {X 0,Y 570.194,Z 462.44,A -85,B 0,C 180,E1 2538.578,E2 2538.578} C_VEL
LIN {X 0,Y 570.123,Z 462.44,A -85,B 0,C 180,E1 2543.472,E2 2543.472} C_VEL
LIN {X 0,Y 569.991,Z 462.44,A -85,B 0,C 180,E1 2548.763,E2 2548.763} C_VEL
LIN {X 0,Y 570.108,Z 462.44,A -85,B 0,C 180,E1 2554.581,E2 2554.581} C_VEL
LIN {X 0,Y 569.983,Z 462.44,A -85,B 0,C 180,E1 2559.613,E2 2559.613} C_VEL
LIN {X 0,Y 569.755,Z 462.44,A -85,B 0,C 180,E1 2565.843,E2 2565.843} C_VEL
LIN {X 0,Y 569.992,Z 462.44,A -85,B 0,C 180,E1 2570.391,E2 2570.391} C_VEL
LIN {X 0,Y 570.239,Z 462.44,A -85,B 0,C 180,E1 2576.11,E2 2576.11} C_VEL
LIN {X 0,Y 570.287,Z 462.44,A -85,B 0,C 180,E1 2578.288,E2 2578.288} C_VEL
LIN {X 0,Y 576.032,Z 478.534,A -85,B 0,C 180,E1 2578.875,E2 2578.875} C_VEL
LIN {X 0,Y 576.125,Z 532.845,A -85,B 0,C 180,E1 2579.828,E2 2579.828} C_VEL
LIN {X 0,Y 575.39,Z 572.213,A -85,B 0,C 180,E1 2581.138,E2 2581.138} C_VEL
LIN {X 0,Y 574.393,Z 608.551,A -85,B 0,C 180,E1 2582.956,E2 2582.956} C_VEL
LIN {X 0,Y 573.271,Z 643.515,A -85,B 0,C 180,E1 2585.365,E2 2585.365} C_VEL
LIN {X 0,Y 572.229,Z 675.15,A -85,B 0,C 180,E1 2588.257,E2 2588.257} C_VEL
LIN {X 0,Y 571.505,Z 702.057,A -85,B 0,C 180,E1 2591.463,E2 2591.463} C_VEL
LIN {X 0,Y 570.978,Z 724.657,A -85,B 0,C 180,E1 2594.988,E2 2594.988} C_VEL
LIN {X 0,Y 570.652,Z 741.41,A -85,B 0,C 180,E1 2598.498,E2 2598.498} C_VEL
LIN {X 0,Y 570.548,Z 754.226,A -85,B 0,C 180,E1 2602.375,E2 2602.375} C_VEL
LIN {X 0,Y 570.472,Z 760.504,A -85,B 0,C 180,E1 2605.433,E2 2605.433} C_VEL
LIN {X 0,Y 570.465,Z 763.613,A -85,B 0,C 180,E1 2608.479,E2 2608.479} C_VEL
LIN {X 0,Y 570.584,Z 763.553,A -85,B 0,C 180,E1 2611.521,E2 2611.521} C_VEL
LIN {X 0,Y 570.668,Z 759.371,A -85,B 0,C 180,E1 2615.194,E2 2615.194} C_VEL
LIN {X 0,Y 570.623,Z 749.574,A -85,B 0,C 180,E1 2619.161,E2 2619.161} C_VEL
LIN {X 0,Y 570.836,Z 734.377,A -85,B 0,C 180,E1 2623.03,E2 2623.03} C_VEL
LIN {X 0,Y 571.199,Z 713.782,A -85,B 0,C 180,E1 2626.755,E2 2626.755} C_VEL
LIN {X 0,Y 571.911,Z 687.102,A -85,B 0,C 180,E1 2630.334,E2 2630.334} C_VEL
LIN {X 0,Y 572.818,Z 657.518,A -85,B 0,C 180,E1 2633.359,E2 2633.359} C_VEL
LIN {X 0,Y 573.88,Z 624.179,A -85,B 0,C 180,E1 2635.964,E2 2635.964} C_VEL
LIN {X 0,Y 574.916,Z 589.398,A -85,B 0,C 180,E1 2637.99,E2 2637.99} C_VEL
LIN {X 0,Y 575.797,Z 552.001,A -85,B 0,C 180,E1 2639.524,E2 2639.524} C_VEL
LIN {X 0,Y 576.344,Z 512.732,A -85,B 0,C 180,E1 2640.507,E2 2640.507} C_VEL
LIN {X 0,Y 575.88,Z 475.993,A -85,B 0,C 180,E1 2641.081,E2 2641.081} C_VEL
LIN {X 0,Y 570.064,Z 462.44,A -85,B 0,C 180,E1 2641.696,E2 2641.696} C_VEL
LIN {X 0,Y 570.13,Z 462.44,A -85,B 0,C 180,E1 2647.649,E2 2647.649} C_VEL
LIN {X 0,Y 569.877,Z 462.44,A -85,B 0,C 180,E1 2654.17,E2 2654.17} C_VEL
LIN {X 0,Y 569.958,Z 462.44,A -85,B 0,C 180,E1 2658.391,E2 2658.391} C_VEL
LIN {X 0,Y 569.96,Z 462.44,A -85,B 0,C 180,E1 2664.242,E2 2664.242} C_VEL
LIN {X 0,Y 570.026,Z 462.44,A -85,B 0,C 180,E1 2669.694,E2 2669.694} C_VEL
LIN {X 0,Y 570.119,Z 462.44,A -85,B 0,C 180,E1 2674.858,E2 2674.858} C_VEL
LIN {X 0,Y 570.227,Z 462.44,A -85,B 0,C 180,E1 2679.81,E2 2679.81} C_VEL
LIN {X 0,Y 570.414,Z 462.44,A -85,B 0,C 180,E1 2686.181,E2 2686.181} C_VEL
LIN {X 0,Y 570.287,Z 462.44,A -85,B 0,C 180,E1 2692.373,E2 2692.373} C_VEL
LIN {X 0,Y 570.398,Z 462.44,A -85,B 0,C 180,E1 2696.958,E2 2696.958} C_VEL
LIN {X 0,Y 570.544,Z 462.44,A -85,B 0,C 180,E1 2701.521,E2 2701.521} C_VEL
LIN {X 0,Y 570.182,Z 462.44,A -85,B 0,C 180,E1 2707.607,E2 2707.607} C_VEL
LIN {X 0,Y 570.265,Z 462.44,A -85,B 0,C 180,E1 2711.018,E2 2711.018} C_VEL
LIN {X 0,Y 566.205,Z 462.44,A -85,B 0,C 180,E1 2712.73,E2 2712.73} C_VEL
LIN {X 0,Y 562.232,Z 462.44,A -85,B 0,C 180,E1 2714.465,E2 2714.465} C_VEL
LIN {X 0,Y 562.249,Z 462.44,A -85,B 0,C 180,E1 2720.491,E2 2720.491} C_VEL
LIN {X 0,Y 562.245,Z 462.44,A -85,B 0,C 180,E1 2725.521,E2 2725.521} C_VEL
LIN {X 0,Y 562.077,Z 462.44,A -85,B 0,C 180,E1 2730.782,E2 2730.782} C_VEL
LIN {X 0,Y 562.105,Z 462.44,A -85,B 0,C 180,E1 2736.338,E2 2736.338} C_VEL
LIN {X 0,Y 562.052,Z 462.44,A -85,B 0,C 180,E1 2742.331,E2 2742.331} C_VEL
LIN {X 0,Y 561.938,Z 462.44,A -85,B 0,C 180,E1 2747.653,E2 2747.653} C_VEL
LIN {X 0,Y 562.027,Z 462.44,A -85,B 0,C 180,E1 2753.12,E2 2753.12} C_VEL
LIN {X 0,Y 571.352,Z 481.87,A -85,B 0,C 180,E1 2754.139,E2 2754.139} C_VEL
LIN {X 0,Y 571.162,Z 532.179,A -85,B 0,C 180,E1 2755.09,E2 2755.09} C_VEL
LIN {X 0,Y 570.122,Z 572.107,A -85,B 0,C 180,E1 2756.425,E2 2756.425} C_VEL
LIN {X 0,Y 568.792,Z 609.403,A -85,B 0,C 180,E1 2758.255,E2 2758.255} C_VEL
LIN {X 0,Y 567.29,Z 645.044,A -85,B 0,C 180,E1 2760.595,E2 2760.595} C_VEL
LIN {X 0,Y 565.78,Z 679.547,A -85,B 0,C 180,E1 2763.538,E2 2763.538} C_VEL
LIN {X 0,Y 564.557,Z 710.344,A -85,B 0,C 180,E1 2766.906,E2 2766.906} C_VEL
LIN {X 0,Y 563.571,Z 736.895,A -85,B 0,C 180,E1 2770.613,E2 2770.613} C_VEL
LIN {X 0,Y 563.008,Z 759.302,A -85,B 0,C 180,E1 2774.713,E2 2774.713} C_VEL
LIN {X 0,Y 562.684,Z 775.918,A -85,B 0,C 180,E1 2778.891,E2 2778.891} C_VEL
LIN {X 0,Y 562.631,Z 785.33,A -85,B 0,C 180,E1 2782.267,E2 2782.267} C_VEL
LIN {X 0,Y 562.725,Z 790.904,A -85,B 0,C 180,E1 2785.37,E2 2785.37} C_VEL
LIN {X 0,Y 562.697,Z 793.657,A -85,B 0,C 180,E1 2788.458,E2 2788.458} C_VEL
LIN {X 0,Y 562.581,Z 792.627,A -85,B 0,C 180,E1 2793.086,E2 2793.086} C_VEL
LIN {X 0,Y 562.722,Z 786.916,A -85,B 0,C 180,E1 2796.955,E2 2796.955} C_VEL
LIN {X 0,Y 562.75,Z 775.756,A -85,B 0,C 180,E1 2801.155,E2 2801.155} C_VEL
LIN {X 0,Y 563.09,Z 759.232,A -85,B 0,C 180,E1 2805.299,E2 2805.299} C_VEL
LIN {X 0,Y 563.605,Z 736.909,A -85,B 0,C 180,E1 2809.384,E2 2809.384} C_VEL
LIN {X 0,Y 564.624,Z 708.673,A -85,B 0,C 180,E1 2813.3,E2 2813.3} C_VEL
LIN {X 0,Y 565.968,Z 676.391,A -85,B 0,C 180,E1 2816.762,E2 2816.762} C_VEL
LIN {X 0,Y 567.494,Z 641.258,A -85,B 0,C 180,E1 2819.688,E2 2819.688} C_VEL
LIN {X 0,Y 569.075,Z 602.247,A -85,B 0,C 180,E1 2822.15,E2 2822.15} C_VEL
LIN {X 0,Y 570.459,Z 562.617,A -85,B 0,C 180,E1 2823.942,E2 2823.942} C_VEL
LIN {X 0,Y 571.375,Z 524.455,A -85,B 0,C 180,E1 2825.091,E2 2825.091} C_VEL
LIN {X 0,Y 571.351,Z 481.889,A -85,B 0,C 180,E1 2825.861,E2 2825.861} C_VEL
LIN {X 0,Y 562.028,Z 462.44,A -85,B 0,C 180,E1 2826.88,E2 2826.88} C_VEL
LIN {X 0,Y 561.94,Z 462.44,A -85,B 0,C 180,E1 2832.347,E2 2832.347} C_VEL
LIN {X 0,Y 562.053,Z 462.44,A -85,B 0,C 180,E1 2837.669,E2 2837.669} C_VEL
LIN {X 0,Y 562.095,Z 462.44,A -85,B 0,C 180,E1 2843.913,E2 2843.913} C_VEL
LIN {X 0,Y 562.11,Z 462.44,A -85,B 0,C 180,E1 2849.539,E2 2849.539} C_VEL
LIN {X 0,Y 562.211,Z 462.44,A -85,B 0,C 180,E1 2854.477,E2 2854.477} C_VEL
LIN {X 0,Y 562.289,Z 462.44,A -85,B 0,C 180,E1 2860.473,E2 2860.473} C_VEL
LIN {X 0,Y 562.162,Z 462.44,A -85,B 0,C 180,E1 2864.376,E2 2864.376} C_VEL
LIN {X 0,Y 562.276,Z 462.44,A -85,B 0,C 180,E1 2870.702,E2 2870.702} C_VEL
LIN {X 0,Y 562.367,Z 462.44,A -85,B 0,C 180,E1 2875.367,E2 2875.367} C_VEL
LIN {X 0,Y 562.407,Z 462.44,A -85,B 0,C 180,E1 2879.999,E2 2879.999} C_VEL
LIN {X 0,Y 562.328,Z 462.44,A -85,B 0,C 180,E1 2884.95,E2 2884.95} C_VEL
LIN {X 0,Y 562.367,Z 462.44,A -85,B 0,C 180,E1 2889.295,E2 2889.295} C_VEL
LIN {X 0,Y 562.289,Z 462.44,A -85,B 0,C 180,E1 2894.208,E2 2894.208} C_VEL
LIN {X 0,Y 562.186,Z 462.44,A -85,B 0,C 180,E1 2899.498,E2 2899.498} C_VEL
LIN {X 0,Y 562.167,Z 462.44,A -85,B 0,C 180,E1 2903.825,E2 2903.825} C_VEL
LIN {X 0,Y 562.061,Z 462.44,A -85,B 0,C 180,E1 2909.001,E2 2909.001} C_VEL
LIN {X 0,Y 562.231,Z 462.44,A -85,B 0,C 180,E1 2914.434,E2 2914.434} C_VEL
LIN {X 0,Y 562.008,Z 462.44,A -85,B 0,C 180,E1 2920.278,E2 2920.278} C_VEL
LIN {X 0,Y 561.817,Z 462.44,A -85,B 0,C 180,E1 2925.515,E2 2925.515} C_VEL
LIN {X 0,Y 562.087,Z 462.44,A -85,B 0,C 180,E1 2931.36,E2 2931.36} C_VEL
LIN {X 0,Y 562.303,Z 462.44,A -85,B 0,C 180,E1 2936.578,E2 2936.578} C_VEL
LIN {X 0,Y 562.376,Z 463.091,A -85,B 0,C 180,E1 2937.804,E2 2937.804} C_VEL
LIN {X 0,Y 569.266,Z 479.779,A -85,B 0,C 180,E1 2938.481,E2 2938.481} C_VEL
LIN {X 0,Y 569.274,Z 533.095,A -85,B 0,C 180,E1 2939.434,E2 2939.434} C_VEL
LIN {X 0,Y 568.436,Z 570.782,A -85,B 0,C 180,E1 2940.687,E2 2940.687} C_VEL
LIN {X 0,Y 567.321,Z 607.088,A -85,B 0,C 180,E1 2942.499,E2 2942.499} C_VEL
LIN {X 0,Y 565.969,Z 642.203,A -85,B 0,C 180,E1 2944.917,E2 2944.917} C_VEL
LIN {X 0,Y 564.719,Z 673.99,A -85,B 0,C 180,E1 2947.828,E2 2947.828} C_VEL
LIN {X 0,Y 563.824,Z 700.9,A -85,B 0,C 180,E1 2951.041,E2 2951.041} C_VEL
LIN {X 0,Y 563.214,Z 722.62,A -85,B 0,C 180,E1 2954.405,E2 2954.405} C_VEL
LIN {X 0,Y 562.789,Z 739.957,A -85,B 0,C 180,E1 2957.965,E2 2957.965} C_VEL
LIN {X 0,Y 562.697,Z 753.262,A -85,B 0,C 180,E1 2961.879,E2 2961.879} C_VEL
LIN {X 0,Y 562.573,Z 760.503,A -85,B 0,C 180,E1 2965.369,E2 2965.369} C_VEL
LIN {X 0,Y 562.563,Z 763.613,A -85,B 0,C 180,E1 2968.458,E2 2968.458} C_VEL
LIN {X 0,Y 562.679,Z 763.553,A -85,B 0,C 180,E1 2971.542,E2 2971.542} C_VEL
LIN {X 0,Y 562.717,Z 759.01,A -85,B 0,C 180,E1 2975.472,E2 2975.472} C_VEL
LIN {X 0,Y 562.745,Z 749.576,A -85,B 0,C 180,E1 2979.29,E2 2979.29} C_VEL
LIN {X 0,Y 562.978,Z 734.381,A -85,B 0,C 180,E1 2983.215,E2 2983.215} C_VEL
LIN {X 0,Y 563.437,Z 713.786,A -85,B 0,C 180,E1 2986.993,E2 2986.993} C_VEL
LIN {X 0,Y 564.261,Z 687.107,A -85,B 0,C 180,E1 2990.622,E2 2990.622} C_VEL
LIN {X 0,Y 565.345,Z 657.527,A -85,B 0,C 180,E1 2993.687,E2 2993.687} C_VEL
LIN {X 0,Y 566.635,Z 624.562,A -85,B 0,C 180,E1 2996.295,E2 2996.295} C_VEL
LIN {X 0,Y 567.846,Z 589.2,A -85,B 0,C 180,E1 2998.381,E2 2998.381} C_VEL
LIN {X 0,Y 568.872,Z 552.544,A -85,B 0,C 180,E1 2999.903,E2 2999.903} C_VEL
LIN {X 0,Y 569.535,Z 513.934,A -85,B 0,C 180,E1 3000.892,E2 3000.892} C_VEL
LIN {X 0,Y 569.045,Z 478.474,A -85,B 0,C 180,E1 3001.461,E2 3001.461} C_VEL
LIN {X 0,Y 562.073,Z 462.44,A -85,B 0,C 180,E1 3002.209,E2 3002.209} C_VEL
LIN {X 0,Y 562.122,Z 462.44,A -85,B 0,C 180,E1 3008.282,E2 3008.282} C_VEL
LIN {X 0,Y 561.966,Z 462.44,A -85,B 0,C 180,E1 3014.47,E2 3014.47} C_VEL
LIN {X 0,Y 561.965,Z 462.44,A -85,B 0,C 180,E1 3019.718,E2 3019.718} C_VEL
LIN {X 0,Y 561.978,Z 462.44,A -85,B 0,C 180,E1 3025.548,E2 3025.548} C_VEL
LIN {X 0,Y 562.053,Z 462.44,A -85,B 0,C 180,E1 3030.998,E2 3030.998} C_VEL
LIN {X 0,Y 562.154,Z 462.44,A -85,B 0,C 180,E1 3036.316,E2 3036.316} C_VEL
LIN {X 0,Y 562.303,Z 462.44,A -85,B 0,C 180,E1 3041.151,E2 3041.151} C_VEL
LIN {X 0,Y 562.47,Z 462.44,A -85,B 0,C 180,E1 3045.982,E2 3045.982} C_VEL
LIN {X 0,Y 562.384,Z 462.44,A -85,B 0,C 180,E1 3052.265,E2 3052.265} C_VEL
LIN {X 0,Y 562.49,Z 462.44,A -85,B 0,C 180,E1 3056.915,E2 3056.915} C_VEL
LIN {X 0,Y 562.633,Z 462.44,A -85,B 0,C 180,E1 3061.543,E2 3061.543} C_VEL
LIN {X 0,Y 562.555,Z 462.44,A -85,B 0,C 180,E1 3066.181,E2 3066.181} C_VEL
LIN {X 0,Y 562.262,Z 462.44,A -85,B 0,C 180,E1 3072.44,E2 3072.44} C_VEL
LIN {X 0,Y 562.232,Z 462.44,A -85,B 0,C 180,E1 3074.465,E2 3074.465} C_VEL
LIN {X 0,Y 558.24,Z 462.44,A -85,B 0,C 180,E1 3076.207,E2 3076.207} C_VEL
LIN {X 0,Y 554.233,Z 462.44,A -85,B 0,C 180,E1 3077.974,E2 3077.974} C_VEL
LIN {X 0,Y 554.27,Z 462.44,A -85,B 0,C 180,E1 3082.483,E2 3082.483} C_VEL
LIN {X 0,Y 554.174,Z 462.44,A -85,B 0,C 180,E1 3087.674,E2 3087.674} C_VEL
LIN {X 0,Y 554.069,Z 462.44,A -85,B 0,C 180,E1 3093.127,E2 3093.127} C_VEL
LIN {X 0,Y 554.143,Z 462.44,A -85,B 0,C 180,E1 3098.931,E2 3098.931} C_VEL
LIN {X 0,Y 554.158,Z 462.44,A -85,B 0,C 180,E1 3104.732,E2 3104.732} C_VEL
LIN {X 0,Y 554.024,Z 462.44,A -85,B 0,C 180,E1 3111.054,E2 3111.054} C_VEL
LIN {X 0,Y 554.174,Z 462.44,A -85,B 0,C 180,E1 3112.506,E2 3112.506} C_VEL
LIN {X 0,Y 561.084,Z 477.332,A -85,B 0,C 180,E1 3113.307,E2 3113.307} C_VEL
LIN {X 0,Y 565.191,Z 485.432,A -85,B 0,C 180,E1 3113.742,E2 3113.742} C_VEL
LIN {X 0,Y 564.641,Z 532.319,A -85,B 0,C 180,E1 3114.631,E2 3114.631} C_VEL
LIN {X 0,Y 563.431,Z 572.81,A -85,B 0,C 180,E1 3116.001,E2 3116.001} C_VEL
LIN {X 0,Y 561.838,Z 611.107,A -85,B 0,C 180,E1 3117.918,E2 3117.918} C_VEL
LIN {X 0,Y 560.096,Z 647.084,A -85,B 0,C 180,E1 3120.343,E2 3120.343} C_VEL
LIN {X 0,Y 558.331,Z 681.845,A -85,B 0,C 180,E1 3123.395,E2 3123.395} C_VEL
LIN {X 0,Y 556.921,Z 711.957,A -85,B 0,C 180,E1 3126.783,E2 3126.783} C_VEL
LIN {X 0,Y 555.793,Z 738.832,A -85,B 0,C 180,E1 3130.658,E2 3130.658} C_VEL
LIN {X 0,Y 555.199,Z 759.128,A -85,B 0,C 180,E1 3134.456,E2 3134.456} C_VEL
LIN {X 0,Y 554.816,Z 775.435,A -85,B 0,C 180,E1 3138.588,E2 3138.588} C_VEL
LIN {X 0,Y 554.742,Z 785.33,A -85,B 0,C 180,E1 3142.156,E2 3142.156} C_VEL
LIN {X 0,Y 554.827,Z 790.904,A -85,B 0,C 180,E1 3145.304,E2 3145.304} C_VEL
LIN {X 0,Y 554.792,Z 793.657,A -85,B 0,C 180,E1 3148.436,E2 3148.436} C_VEL
LIN {X 0,Y 554.691,Z 792.627,A -85,B 0,C 180,E1 3153.13,E2 3153.13} C_VEL
LIN {X 0,Y 554.831,Z 786.916,A -85,B 0,C 180,E1 3157.054,E2 3157.054} C_VEL
LIN {X 0,Y 554.886,Z 776.774,A -85,B 0,C 180,E1 3161.012,E2 3161.012} C_VEL
LIN {X 0,Y 555.24,Z 760.305,A -85,B 0,C 180,E1 3165.286,E2 3165.286} C_VEL
LIN {X 0,Y 555.828,Z 738.848,A -85,B 0,C 180,E1 3169.338,E2 3169.338} C_VEL
LIN {X 0,Y 556.961,Z 711.964,A -85,B 0,C 180,E1 3173.215,E2 3173.215} C_VEL
LIN {X 0,Y 558.445,Z 680.45,A -85,B 0,C 180,E1 3176.744,E2 3176.744} C_VEL
LIN {X 0,Y 560.208,Z 644.999,A -85,B 0,C 180,E1 3179.818,E2 3179.818} C_VEL
LIN {X 0,Y 561.949,Z 607.547,A -85,B 0,C 180,E1 3182.29,E2 3182.29} C_VEL
LIN {X 0,Y 563.565,Z 569.47,A -85,B 0,C 180,E1 3184.13,E2 3184.13} C_VEL
LIN {X 0,Y 564.786,Z 529.301,A -85,B 0,C 180,E1 3185.445,E2 3185.445} C_VEL
LIN {X 0,Y 564.789,Z 484.631,A -85,B 0,C 180,E1 3186.301,E2 3186.301} C_VEL
LIN {X 0,Y 554.23,Z 463.673,A -85,B 0,C 180,E1 3187.441,E2 3187.441} C_VEL
LIN {X 0,Y 554.126,Z 462.44,A -85,B 0,C 180,E1 3187.596,E2 3187.596} C_VEL
LIN {X 0,Y 554.065,Z 462.44,A -85,B 0,C 180,E1 3193.094,E2 3193.094} C_VEL
LIN {X 0,Y 554.129,Z 462.44,A -85,B 0,C 180,E1 3199.025,E2 3199.025} C_VEL
LIN {X 0,Y 554.1,Z 462.44,A -85,B 0,C 180,E1 3205.063,E2 3205.063} C_VEL
LIN {X 0,Y 554.182,Z 462.44,A -85,B 0,C 180,E1 3210.963,E2 3210.963} C_VEL
LIN {X 0,Y 554.242,Z 462.44,A -85,B 0,C 180,E1 3215.811,E2 3215.811} C_VEL
LIN {X 0,Y 554.397,Z 462.44,A -85,B 0,C 180,E1 3220.87,E2 3220.87} C_VEL
LIN {X 0,Y 554.085,Z 462.44,A -85,B 0,C 180,E1 3225.763,E2 3225.763} C_VEL
LIN {X 0,Y 554.365,Z 462.44,A -85,B 0,C 180,E1 3230.568,E2 3230.568} C_VEL
LIN {X 0,Y 554.49,Z 462.44,A -85,B 0,C 180,E1 3235.301,E2 3235.301} C_VEL
LIN {X 0,Y 554.506,Z 462.44,A -85,B 0,C 180,E1 3239.999,E2 3239.999} C_VEL
LIN {X 0,Y 554.483,Z 462.44,A -85,B 0,C 180,E1 3244.698,E2 3244.698} C_VEL
LIN {X 0,Y 554.341,Z 462.44,A -85,B 0,C 180,E1 3250.483,E2 3250.483} C_VEL
LIN {X 0,Y 554.233,Z 462.44,A -85,B 0,C 180,E1 3255.852,E2 3255.852} C_VEL
LIN {X 0,Y 554.263,Z 462.44,A -85,B 0,C 180,E1 3261.75,E2 3261.75} C_VEL
LIN {X 0,Y 554.149,Z 462.44,A -85,B 0,C 180,E1 3267.673,E2 3267.673} C_VEL
LIN {X 0,Y 554.26,Z 462.44,A -85,B 0,C 180,E1 3273.112,E2 3273.112} C_VEL
LIN {X 0,Y 554.126,Z 462.44,A -85,B 0,C 180,E1 3278.931,E2 3278.931} C_VEL
LIN {X 0,Y 553.904,Z 462.44,A -85,B 0,C 180,E1 3284.706,E2 3284.706} C_VEL
LIN {X 0,Y 554.098,Z 462.44,A -85,B 0,C 180,E1 3289.909,E2 3289.909} C_VEL
LIN {X 0,Y 554.385,Z 462.44,A -85,B 0,C 180,E1 3295.009,E2 3295.009} C_VEL
LIN {X 0,Y 554.407,Z 462.44,A -85,B 0,C 180,E1 3297.266,E2 3297.266} C_VEL
LIN {X 0,Y 562.569,Z 483.49,A -85,B 0,C 180,E1 3298.117,E2 3298.117} C_VEL
LIN {X 0,Y 562.474,Z 532.896,A -85,B 0,C 180,E1 3299.019,E2 3299.019} C_VEL
LIN {X 0,Y 561.44,Z 571.763,A -85,B 0,C 180,E1 3300.331,E2 3300.331} C_VEL
LIN {X 0,Y 560.13,Z 608.499,A -85,B 0,C 180,E1 3302.207,E2 3302.207} C_VEL
LIN {X 0,Y 558.595,Z 642.902,A -85,B 0,C 180,E1 3304.623,E2 3304.623} C_VEL
LIN {X 0,Y 557.128,Z 675.137,A -85,B 0,C 180,E1 3307.636,E2 3307.636} C_VEL
LIN {X 0,Y 556.094,Z 702.049,A -85,B 0,C 180,E1 3310.929,E2 3310.929} C_VEL
LIN {X 0,Y 555.369,Z 724.038,A -85,B 0,C 180,E1 3314.442,E2 3314.442} C_VEL
LIN {X 0,Y 554.918,Z 741.499,A -85,B 0,C 180,E1 3318.191,E2 3318.191} C_VEL
LIN {X 0,Y 554.823,Z 753.26,A -85,B 0,C 180,E1 3321.763,E2 3321.763} C_VEL
LIN {X 0,Y 554.685,Z 760.502,A -85,B 0,C 180,E1 3325.303,E2 3325.303} C_VEL
LIN {X 0,Y 554.66,Z 763.613,A -85,B 0,C 180,E1 3328.436,E2 3328.436} C_VEL
LIN {X 0,Y 554.774,Z 763.554,A -85,B 0,C 180,E1 3331.564,E2 3331.564} C_VEL
LIN {X 0,Y 554.806,Z 759.012,A -85,B 0,C 180,E1 3335.55,E2 3335.55} C_VEL
LIN {X 0,Y 554.848,Z 749.578,A -85,B 0,C 180,E1 3339.424,E2 3339.424} C_VEL
LIN {X 0,Y 555.157,Z 734.385,A -85,B 0,C 180,E1 3343.405,E2 3343.405} C_VEL
LIN {X 0,Y 555.706,Z 713.791,A -85,B 0,C 180,E1 3347.236,E2 3347.236} C_VEL
LIN {X 0,Y 556.648,Z 687.112,A -85,B 0,C 180,E1 3350.917,E2 3350.917} C_VEL
LIN {X 0,Y 557.917,Z 657.537,A -85,B 0,C 180,E1 3354.022,E2 3354.022} C_VEL
LIN {X 0,Y 559.38,Z 624.965,A -85,B 0,C 180,E1 3356.635,E2 3356.635} C_VEL
LIN {X 0,Y 560.817,Z 589.217,A -85,B 0,C 180,E1 3358.769,E2 3358.769} C_VEL
LIN {X 0,Y 562.009,Z 552.932,A -85,B 0,C 180,E1 3360.293,E2 3360.293} C_VEL
LIN {X 0,Y 562.773,Z 515.054,A -85,B 0,C 180,E1 3361.286,E2 3361.286} C_VEL
LIN {X 0,Y 562.248,Z 480.769,A -85,B 0,C 180,E1 3361.853,E2 3361.853} C_VEL
LIN {X 0,Y 554.11,Z 462.44,A -85,B 0,C 180,E1 3362.66,E2 3362.66} C_VEL
LIN {X 0,Y 554.174,Z 462.44,A -85,B 0,C 180,E1 3368.933,E2 3368.933} C_VEL
LIN {X 0,Y 554.098,Z 462.44,A -85,B 0,C 180,E1 3375.274,E2 3375.274} C_VEL
LIN {X 0,Y 554.048,Z 462.44,A -85,B 0,C 180,E1 3381.063,E2 3381.063} C_VEL
LIN {X 0,Y 554.057,Z 462.44,A -85,B 0,C 180,E1 3386.874,E2 3386.874} C_VEL
LIN {X 0,Y 554.163,Z 462.44,A -85,B 0,C 180,E1 3392.327,E2 3392.327} C_VEL
LIN {X 0,Y 554.273,Z 462.44,A -85,B 0,C 180,E1 3398.248,E2 3398.248} C_VEL
LIN {X 0,Y 554.416,Z 462.44,A -85,B 0,C 180,E1 3404.154,E2 3404.154} C_VEL
LIN {X 0,Y 554.401,Z 462.44,A -85,B 0,C 180,E1 3409.484,E2 3409.484} C_VEL
LIN {X 0,Y 554.513,Z 462.44,A -85,B 0,C 180,E1 3415.303,E2 3415.303} C_VEL
LIN {X 0,Y 554.722,Z 462.44,A -85,B 0,C 180,E1 3421.565,E2 3421.565} C_VEL
LIN {X 0,Y 554.37,Z 462.44,A -85,B 0,C 180,E1 3427.849,E2 3427.849} C_VEL
LIN {X 0,Y 554.341,Z 462.44,A -85,B 0,C 180,E1 3432.621,E2 3432.621} C_VEL
LIN {X 0,Y 554.233,Z 462.44,A -85,B 0,C 180,E1 3437.974,E2 3437.974} C_VEL
LIN {X 0,Y 550.32,Z 462.44,A -85,B 0,C 180,E1 3439.739,E2 3439.739} C_VEL
LIN {X 0,Y 546.342,Z 462.44,A -85,B 0,C 180,E1 3441.53,E2 3441.53} C_VEL
LIN {X 0,Y 546.323,Z 462.44,A -85,B 0,C 180,E1 3446.321,E2 3446.321} C_VEL
LIN {X 0,Y 546.169,Z 462.44,A -85,B 0,C 180,E1 3451.782,E2 3451.782} C_VEL
LIN {X 0,Y 546.224,Z 462.44,A -85,B 0,C 180,E1 3457.574,E2 3457.574} C_VEL
LIN {X 0,Y 546.214,Z 462.44,A -85,B 0,C 180,E1 3463.885,E2 3463.885} C_VEL
LIN {X 0,Y 546.108,Z 462.44,A -85,B 0,C 180,E1 3470.38,E2 3470.38} C_VEL
LIN {X 0,Y 546.166,Z 462.44,A -85,B 0,C 180,E1 3471.862,E2 3471.862} C_VEL
LIN {X 0,Y 557.287,Z 485.368,A -85,B 0,C 180,E1 3473.142,E2 3473.142} C_VEL
LIN {X 0,Y 558.895,Z 490.03,A -85,B 0,C 180,E1 3473.339,E2 3473.339} C_VEL
LIN {X 0,Y 558.115,Z 534.03,A -85,B 0,C 180,E1 3474.206,E2 3474.206} C_VEL
LIN {X 0,Y 556.716,Z 575.1,A -85,B 0,C 180,E1 3475.639,E2 3475.639} C_VEL
LIN {X 0,Y 554.889,Z 613.939,A -85,B 0,C 180,E1 3477.642,E2 3477.642} C_VEL
LIN {X 0,Y 552.801,Z 651.152,A -85,B 0,C 180,E1 3480.245,E2 3480.245} C_VEL
LIN {X 0,Y 550.787,Z 686.029,A -85,B 0,C 180,E1 3483.441,E2 3483.441} C_VEL
LIN {X 0,Y 549.143,Z 716.782,A -85,B 0,C 180,E1 3487.079,E2 3487.079} C_VEL
LIN {X 0,Y 547.931,Z 742.793,A -85,B 0,C 180,E1 3491.053,E2 3491.053} C_VEL
LIN {X 0,Y 547.316,Z 761.488,A -85,B 0,C 180,E1 3494.764,E2 3494.764} C_VEL
LIN {X 0,Y 546.917,Z 776.773,A -85,B 0,C 180,E1 3498.826,E2 3498.826} C_VEL
LIN {X 0,Y 546.814,Z 786.916,A -85,B 0,C 180,E1 3502.842,E2 3502.842} C_VEL
LIN {X 0,Y 546.779,Z 792.627,A -85,B 0,C 180,E1 3506.825,E2 3506.825} C_VEL
LIN {X 0,Y 546.802,Z 794,A -85,B 0,C 180,E1 3510,E2 3510} C_VEL
LIN {X 0,Y 546.798,Z 790.905,A -85,B 0,C 180,E1 3514.765,E2 3514.765} C_VEL
LIN {X 0,Y 546.871,Z 783.403,A -85,B 0,C 180,E1 3518.759,E2 3518.759} C_VEL
LIN {X 0,Y 547.053,Z 771.303,A -85,B 0,C 180,E1 3522.793,E2 3522.793} C_VEL
LIN {X 0,Y 547.625,Z 753.017,A -85,B 0,C 180,E1 3527.048,E2 3527.048} C_VEL
LIN {X 0,Y 548.606,Z 728.782,A -85,B 0,C 180,E1 3531.222,E2 3531.222} C_VEL
LIN {X 0,Y 550.116,Z 699.197,A -85,B 0,C 180,E1 3535.118,E2 3535.118} C_VEL
LIN {X 0,Y 552.051,Z 664.313,A -85,B 0,C 180,E1 3538.647,E2 3538.647} C_VEL
LIN {X 0,Y 554.082,Z 626.911,A -85,B 0,C 180,E1 3541.541,E2 3541.541} C_VEL
LIN {X 0,Y 556.146,Z 585.96,A -85,B 0,C 180,E1 3543.873,E2 3543.873} C_VEL
LIN {X 0,Y 557.799,Z 542.378,A -85,B 0,C 180,E1 3545.564,E2 3545.564} C_VEL
LIN {X 0,Y 558.993,Z 497.093,A -85,B 0,C 180,E1 3546.543,E2 3546.543} C_VEL
LIN {X 0,Y 558.356,Z 487.245,A -85,B 0,C 180,E1 3546.746,E2 3546.746} C_VEL
LIN {X 0,Y 546.23,Z 463.445,A -85,B 0,C 180,E1 3548.09,E2 3548.09} C_VEL
LIN {X 0,Y 546.138,Z 462.44,A -85,B 0,C 180,E1 3548.3,E2 3548.3} C_VEL
LIN {X 0,Y 546.161,Z 462.44,A -85,B 0,C 180,E1 3553.885,E2 3553.885} C_VEL
LIN {X 0,Y 546.198,Z 462.44,A -85,B 0,C 180,E1 3558.459,E2 3558.459} C_VEL
LIN {X 0,Y 546.14,Z 462.44,A -85,B 0,C 180,E1 3564.398,E2 3564.398} C_VEL
LIN {X 0,Y 546.175,Z 462.44,A -85,B 0,C 180,E1 3570.069,E2 3570.069} C_VEL
LIN {X 0,Y 546.32,Z 462.44,A -85,B 0,C 180,E1 3576.149,E2 3576.149} C_VEL
LIN {X 0,Y 546.496,Z 462.44,A -85,B 0,C 180,E1 3582.257,E2 3582.257} C_VEL
LIN {X 0,Y 546.433,Z 462.44,A -85,B 0,C 180,E1 3588.816,E2 3588.816} C_VEL
LIN {X 0,Y 546.613,Z 462.44,A -85,B 0,C 180,E1 3595.233,E2 3595.233} C_VEL
LIN {X 0,Y 546.606,Z 462.44,A -85,B 0,C 180,E1 3599.999,E2 3599.999} C_VEL
LIN {X 0,Y 546.584,Z 462.44,A -85,B 0,C 180,E1 3604.766,E2 3604.766} C_VEL
LIN {X 0,Y 546.52,Z 462.44,A -85,B 0,C 180,E1 3609.567,E2 3609.567} C_VEL
LIN {X 0,Y 546.471,Z 462.44,A -85,B 0,C 180,E1 3614.437,E2 3614.437} C_VEL
LIN {X 0,Y 546.385,Z 462.44,A -85,B 0,C 180,E1 3619.575,E2 3619.575} C_VEL
LIN {X 0,Y 546.289,Z 462.44,A -85,B 0,C 180,E1 3624.562,E2 3624.562} C_VEL
LIN {X 0,Y 546.175,Z 462.44,A -85,B 0,C 180,E1 3630.751,E2 3630.751} C_VEL
LIN {X 0,Y 546.227,Z 462.44,A -85,B 0,C 180,E1 3636.498,E2 3636.498} C_VEL
LIN {X 0,Y 546.132,Z 462.44,A -85,B 0,C 180,E1 3641.705,E2 3641.705} C_VEL
LIN {X 0,Y 546.135,Z 462.44,A -85,B 0,C 180,E1 3648.457,E2 3648.457} C_VEL
LIN {X 0,Y 546.37,Z 462.44,A -85,B 0,C 180,E1 3654.411,E2 3654.411} C_VEL
LIN {X 0,Y 546.481,Z 462.702,A -85,B 0,C 180,E1 3656.745,E2 3656.745} C_VEL
LIN {X 0,Y 555.777,Z 483.716,A -85,B 0,C 180,E1 3657.685,E2 3657.685} C_VEL
LIN {X 0,Y 555.697,Z 532.746,A -85,B 0,C 180,E1 3658.595,E2 3658.595} C_VEL
LIN {X 0,Y 554.502,Z 571.108,A -85,B 0,C 180,E1 3659.893,E2 3659.893} C_VEL
LIN {X 0,Y 552.992,Z 608.406,A -85,B 0,C 180,E1 3661.812,E2 3661.812} C_VEL
LIN {X 0,Y 551.261,Z 643.086,A -85,B 0,C 180,E1 3664.278,E2 3664.278} C_VEL
LIN {X 0,Y 549.624,Z 675.13,A -85,B 0,C 180,E1 3667.314,E2 3667.314} C_VEL
LIN {X 0,Y 548.388,Z 702.045,A -85,B 0,C 180,E1 3670.651,E2 3670.651} C_VEL
LIN {X 0,Y 547.565,Z 725.024,A -85,B 0,C 180,E1 3674.4,E2 3674.4} C_VEL
LIN {X 0,Y 547.056,Z 741.497,A -85,B 0,C 180,E1 3678.019,E2 3678.019} C_VEL
LIN {X 0,Y 546.952,Z 753.259,A -85,B 0,C 180,E1 3681.643,E2 3681.643} C_VEL
LIN {X 0,Y 546.784,Z 760.733,A -85,B 0,C 180,E1 3685.388,E2 3685.388} C_VEL
LIN {X 0,Y 546.758,Z 763.612,A -85,B 0,C 180,E1 3688.413,E2 3688.413} C_VEL
LIN {X 0,Y 546.869,Z 763.554,A -85,B 0,C 180,E1 3691.587,E2 3691.587} C_VEL
LIN {X 0,Y 546.912,Z 759.147,A -85,B 0,C 180,E1 3695.561,E2 3695.561} C_VEL
LIN {X 0,Y 546.985,Z 749.58,A -85,B 0,C 180,E1 3699.561,E2 3699.561} C_VEL
LIN {X 0,Y 547.33,Z 734.389,A -85,B 0,C 180,E1 3703.6,E2 3703.6} C_VEL
LIN {X 0,Y 547.965,Z 713.842,A -85,B 0,C 180,E1 3707.48,E2 3707.48} C_VEL
LIN {X 0,Y 549.068,Z 687.117,A -85,B 0,C 180,E1 3711.22,E2 3711.22} C_VEL
LIN {X 0,Y 550.479,Z 657.546,A -85,B 0,C 180,E1 3714.367,E2 3714.367} C_VEL
LIN {X 0,Y 552.143,Z 625.018,A -85,B 0,C 180,E1 3717.009,E2 3717.009} C_VEL
LIN {X 0,Y 553.753,Z 590.765,A -85,B 0,C 180,E1 3719.091,E2 3719.091} C_VEL
LIN {X 0,Y 555.128,Z 553.988,A -85,B 0,C 180,E1 3720.673,E2 3720.673} C_VEL
LIN {X 0,Y 556.023,Z 515.897,A -85,B 0,C 180,E1 3721.696,E2 3721.696} C_VEL
LIN {X 0,Y 555.831,Z 484.017,A -85,B 0,C 180,E1 3722.217,E2 3722.217} C_VEL
LIN {X 0,Y 546.168,Z 462.44,A -85,B 0,C 180,E1 3723.272,E2 3723.272} C_VEL
LIN {X 0,Y 546.253,Z 462.44,A -85,B 0,C 180,E1 3729.103,E2 3729.103} C_VEL
LIN {X 0,Y 546.099,Z 462.44,A -85,B 0,C 180,E1 3733.881,E2 3733.881} C_VEL
LIN {X 0,Y 546.162,Z 462.44,A -85,B 0,C 180,E1 3738.463,E2 3738.463} C_VEL
LIN {X 0,Y 546.106,Z 462.44,A -85,B 0,C 180,E1 3744.397,E2 3744.397} C_VEL
LIN {X 0,Y 546.171,Z 462.44,A -85,B 0,C 180,E1 3750.071,E2 3750.071} C_VEL
LIN {X 0,Y 546.311,Z 462.44,A -85,B 0,C 180,E1 3756.151,E2 3756.151} C_VEL
LIN {X 0,Y 546.451,Z 462.44,A -85,B 0,C 180,E1 3760.583,E2 3760.583} C_VEL
LIN {X 0,Y 546.666,Z 462.44,A -85,B 0,C 180,E1 3765.793,E2 3765.793} C_VEL
LIN {X 0,Y 546.559,Z 462.44,A -85,B 0,C 180,E1 3772.04,E2 3772.04} C_VEL
LIN {X 0,Y 546.695,Z 462.44,A -85,B 0,C 180,E1 3776.826,E2 3776.826} C_VEL
LIN {X 0,Y 546.813,Z 462.44,A -85,B 0,C 180,E1 3781.587,E2 3781.587} C_VEL
LIN {X 0,Y 546.72,Z 462.44,A -85,B 0,C 180,E1 3786.36,E2 3786.36} C_VEL
LIN {X 0,Y 546.422,Z 462.44,A -85,B 0,C 180,E1 3792.807,E2 3792.807} C_VEL
LIN {X 0,Y 546.325,Z 462.44,A -85,B 0,C 180,E1 3797.965,E2 3797.965} C_VEL
LIN {X 0,Y 546.342,Z 462.44,A -85,B 0,C 180,E1 3801.53,E2 3801.53} C_VEL
LIN {X 0,Y 542.355,Z 462.44,A -85,B 0,C 180,E1 3803.319,E2 3803.319} C_VEL
LIN {X 0,Y 538.401,Z 462.44,A -85,B 0,C 180,E1 3805.134,E2 3805.134} C_VEL
LIN {X 0,Y 538.266,Z 462.44,A -85,B 0,C 180,E1 3810.417,E2 3810.417} C_VEL
LIN {X 0,Y 538.245,Z 462.44,A -85,B 0,C 180,E1 3816.206,E2 3816.206} C_VEL
LIN {X 0,Y 538.216,Z 462.44,A -85,B 0,C 180,E1 3822.463,E2 3822.463} C_VEL
LIN {X 0,Y 538.148,Z 462.44,A -85,B 0,C 180,E1 3827.525,E2 3827.525} C_VEL
LIN {X 0,Y 538.251,Z 463.059,A -85,B 0,C 180,E1 3831.235,E2 3831.235} C_VEL
LIN {X 0,Y 552.545,Z 491.18,A -85,B 0,C 180,E1 3832.866,E2 3832.866} C_VEL
LIN {X 0,Y 551.674,Z 534.521,A -85,B 0,C 180,E1 3833.737,E2 3833.737} C_VEL
LIN {X 0,Y 550.143,Z 574.409,A -85,B 0,C 180,E1 3835.135,E2 3835.135} C_VEL
LIN {X 0,Y 548.09,Z 612.933,A -85,B 0,C 180,E1 3837.127,E2 3837.127} C_VEL
LIN {X 0,Y 545.757,Z 650.246,A -85,B 0,C 180,E1 3839.746,E2 3839.746} C_VEL
LIN {X 0,Y 543.556,Z 684.314,A -85,B 0,C 180,E1 3842.876,E2 3842.876} C_VEL
LIN {X 0,Y 541.783,Z 713.572,A -85,B 0,C 180,E1 3846.313,E2 3846.313} C_VEL
LIN {X 0,Y 540.393,Z 739.217,A -85,B 0,C 180,E1 3850.151,E2 3850.151} C_VEL
LIN {X 0,Y 539.604,Z 759.715,A -85,B 0,C 180,E1 3854.122,E2 3854.122} C_VEL
LIN {X 0,Y 539.114,Z 775.435,A -85,B 0,C 180,E1 3858.251,E2 3858.251} C_VEL
LIN {X 0,Y 538.981,Z 785.33,A -85,B 0,C 180,E1 3861.925,E2 3861.925} C_VEL
LIN {X 0,Y 539.075,Z 790.904,A -85,B 0,C 180,E1 3865.166,E2 3865.166} C_VEL
LIN {X 0,Y 538.995,Z 793.657,A -85,B 0,C 180,E1 3868.39,E2 3868.39} C_VEL
LIN {X 0,Y 538.9,Z 792.628,A -85,B 0,C 180,E1 3873.221,E2 3873.221} C_VEL
LIN {X 0,Y 539.031,Z 786.917,A -85,B 0,C 180,E1 3877.262,E2 3877.262} C_VEL
LIN {X 0,Y 539.108,Z 776.773,A -85,B 0,C 180,E1 3881.338,E2 3881.338} C_VEL
LIN {X 0,Y 539.586,Z 759.713,A -85,B 0,C 180,E1 3885.878,E2 3885.878} C_VEL
LIN {X 0,Y 540.525,Z 736.954,A -85,B 0,C 180,E1 3890.239,E2 3890.239} C_VEL
LIN {X 0,Y 542.05,Z 708.669,A -85,B 0,C 180,E1 3894.332,E2 3894.332} C_VEL
LIN {X 0,Y 544.054,Z 677.141,A -85,B 0,C 180,E1 3897.858,E2 3897.858} C_VEL
LIN {X 0,Y 546.446,Z 640.068,A -85,B 0,C 180,E1 3901.046,E2 3901.046} C_VEL
LIN {X 0,Y 548.769,Z 601.167,A -85,B 0,C 180,E1 3903.555,E2 3903.555} C_VEL
LIN {X 0,Y 550.793,Z 560.857,A -85,B 0,C 180,E1 3905.406,E2 3905.406} C_VEL
LIN {X 0,Y 552.087,Z 524.948,A -85,B 0,C 180,E1 3906.498,E2 3906.498} C_VEL
LIN {X 0,Y 552.113,Z 490.375,A -85,B 0,C 180,E1 3907.181,E2 3907.181} C_VEL
LIN {X 0,Y 538.253,Z 463.063,A -85,B 0,C 180,E1 3908.765,E2 3908.765} C_VEL
LIN {X 0,Y 538.213,Z 462.44,A -85,B 0,C 180,E1 3914.694,E2 3914.694} C_VEL
LIN {X 0,Y 538.235,Z 462.44,A -85,B 0,C 180,E1 3919.687,E2 3919.687} C_VEL
LIN {X 0,Y 538.203,Z 462.44,A -85,B 0,C 180,E1 3925.763,E2 3925.763} C_VEL
LIN {X 0,Y 538.277,Z 462.44,A -85,B 0,C 180,E1 3931.435,E2 3931.435} C_VEL
LIN {X 0,Y 538.408,Z 462.44,A -85,B 0,C 180,E1 3936.816,E2 3936.816} C_VEL
LIN {X 0,Y 538.573,Z 462.44,A -85,B 0,C 180,E1 3941.987,E2 3941.987} C_VEL
LIN {X 0,Y 538.508,Z 462.44,A -85,B 0,C 180,E1 3948.649,E2 3948.649} C_VEL
LIN {X 0,Y 538.71,Z 462.44,A -85,B 0,C 180,E1 3955.163,E2 3955.163} C_VEL
LIN {X 0,Y 538.724,Z 462.44,A -85,B 0,C 180,E1 3959.999,E2 3959.999} C_VEL
LIN {X 0,Y 538.672,Z 462.44,A -85,B 0,C 180,E1 3964.836,E2 3964.836} C_VEL
LIN {X 0,Y 538.542,Z 462.44,A -85,B 0,C 180,E1 3970.25,E2 3970.25} C_VEL
LIN {X 0,Y 538.527,Z 462.44,A -85,B 0,C 180,E1 3974.655,E2 3974.655} C_VEL
LIN {X 0,Y 538.478,Z 462.44,A -85,B 0,C 180,E1 3979.717,E2 3979.717} C_VEL
LIN {X 0,Y 538.288,Z 462.44,A -85,B 0,C 180,E1 3985.826,E2 3985.826} C_VEL
LIN {X 0,Y 538.279,Z 462.44,A -85,B 0,C 180,E1 3990.414,E2 3990.414} C_VEL
LIN {X 0,Y 538.328,Z 462.44,A -85,B 0,C 180,E1 3996.198,E2 3996.198} C_VEL
LIN {X 0,Y 538.098,Z 462.44,A -85,B 0,C 180,E1 4002.472,E2 4002.472} C_VEL
LIN {X 0,Y 538.095,Z 462.44,A -85,B 0,C 180,E1 4007.52,E2 4007.52} C_VEL
LIN {X 0,Y 538.439,Z 462.44,A -85,B 0,C 180,E1 4013.805,E2 4013.805} C_VEL
LIN {X 0,Y 538.557,Z 463.156,A -85,B 0,C 180,E1 4016.198,E2 4016.198} C_VEL
LIN {X 0,Y 549.174,Z 486.587,A -85,B 0,C 180,E1 4017.293,E2 4017.293} C_VEL
LIN {X 0,Y 548.899,Z 534.287,A -85,B 0,C 180,E1 4018.207,E2 4018.207} C_VEL
LIN {X 0,Y 547.584,Z 571.685,A -85,B 0,C 180,E1 4019.5,E2 4019.5} C_VEL
LIN {X 0,Y 545.92,Z 607.956,A -85,B 0,C 180,E1 4021.384,E2 4021.384} C_VEL
LIN {X 0,Y 543.995,Z 642.548,A -85,B 0,C 180,E1 4023.862,E2 4023.862} C_VEL
LIN {X 0,Y 542.265,Z 673.199,A -85,B 0,C 180,E1 4026.771,E2 4026.771} C_VEL
LIN {X 0,Y 540.774,Z 700.678,A -85,B 0,C 180,E1 4030.17,E2 4030.17} C_VEL
LIN {X 0,Y 539.774,Z 723.709,A -85,B 0,C 180,E1 4033.918,E2 4033.918} C_VEL
LIN {X 0,Y 539.202,Z 741.495,A -85,B 0,C 180,E1 4037.842,E2 4037.842} C_VEL
LIN {X 0,Y 539.051,Z 753.257,A -85,B 0,C 180,E1 4041.52,E2 4041.52} C_VEL
LIN {X 0,Y 538.914,Z 760.501,A -85,B 0,C 180,E1 4045.165,E2 4045.165} C_VEL
LIN {X 0,Y 538.874,Z 763.612,A -85,B 0,C 180,E1 4048.39,E2 4048.39} C_VEL
LIN {X 0,Y 538.978,Z 763.555,A -85,B 0,C 180,E1 4051.61,E2 4051.61} C_VEL
LIN {X 0,Y 539.004,Z 759.148,A -85,B 0,C 180,E1 4055.642,E2 4055.642} C_VEL
LIN {X 0,Y 539.086,Z 749.583,A -85,B 0,C 180,E1 4059.702,E2 4059.702} C_VEL
LIN {X 0,Y 539.482,Z 734.445,A -85,B 0,C 180,E1 4063.79,E2 4063.79} C_VEL
LIN {X 0,Y 540.217,Z 714.256,A -85,B 0,C 180,E1 4067.668,E2 4067.668} C_VEL
LIN {X 0,Y 541.491,Z 687.288,A -85,B 0,C 180,E1 4071.511,E2 4071.511} C_VEL
LIN {X 0,Y 543.08,Z 657.555,A -85,B 0,C 180,E1 4074.722,E2 4074.722} C_VEL
LIN {X 0,Y 545.033,Z 623.569,A -85,B 0,C 180,E1 4077.498,E2 4077.498} C_VEL
LIN {X 0,Y 546.838,Z 588.416,A -85,B 0,C 180,E1 4079.621,E2 4079.621} C_VEL
LIN {X 0,Y 548.312,Z 552.861,A -85,B 0,C 180,E1 4081.137,E2 4081.137} C_VEL
LIN {X 0,Y 549.353,Z 514.09,A -85,B 0,C 180,E1 4082.159,E2 4082.159} C_VEL
LIN {X 0,Y 548.857,Z 486.079,A -85,B 0,C 180,E1 4082.646,E2 4082.646} C_VEL
LIN {X 0,Y 538.258,Z 462.44,A -85,B 0,C 180,E1 4083.791,E2 4083.791} C_VEL
LIN {X 0,Y 538.328,Z 462.44,A -85,B 0,C 180,E1 4088.228,E2 4088.228} C_VEL
LIN {X 0,Y 538.122,Z 462.44,A -85,B 0,C 180,E1 4094.703,E2 4094.703} C_VEL
LIN {X 0,Y 538.173,Z 462.44,A -85,B 0,C 180,E1 4099.684,E2 4099.684} C_VEL
LIN {X 0,Y 538.167,Z 462.44,A -85,B 0,C 180,E1 4105.763,E2 4105.763} C_VEL
LIN {X 0,Y 538.27,Z 462.44,A -85,B 0,C 180,E1 4111.437,E2 4111.437} C_VEL
LIN {X 0,Y 538.397,Z 462.44,A -85,B 0,C 180,E1 4116.818,E2 4116.818} C_VEL
LIN {X 0,Y 538.542,Z 462.44,A -85,B 0,C 180,E1 4121.988,E2 4121.988} C_VEL
LIN {X 0,Y 538.666,Z 462.44,A -85,B 0,C 180,E1 4127.007,E2 4127.007} C_VEL
LIN {X 0,Y 538.645,Z 462.44,A -85,B 0,C 180,E1 4131.922,E2 4131.922} C_VEL
LIN {X 0,Y 538.791,Z 462.44,A -85,B 0,C 180,E1 4136.779,E2 4136.779} C_VEL
LIN {X 0,Y 538.922,Z 462.44,A -85,B 0,C 180,E1 4141.611,E2 4141.611} C_VEL
LIN {X 0,Y 538.79,Z 462.44,A -85,B 0,C 180,E1 4146.454,E2 4146.454} C_VEL
LIN {X 0,Y 538.526,Z 462.44,A -85,B 0,C 180,E1 4152.998,E2 4152.998} C_VEL
LIN {X 0,Y 538.449,Z 462.44,A -85,B 0,C 180,E1 4158.017,E2 4158.017} C_VEL
LIN {X 0,Y 538.423,Z 462.44,A -85,B 0,C 180,E1 4163.183,E2 4163.183} C_VEL
LIN {X 0,Y 538.401,Z 462.44,A -85,B 0,C 180,E1 4165.134,E2 4165.134} C_VEL
LIN {X 0,Y 537.084,Z 462.44,A -85,B 0,C 180,E1 4166.056,E2 4166.056} C_VEL
LIN {X 0,Y 530.423,Z 462.44,A -85,B 0,C 180,E1 4168.566,E2 4168.566} C_VEL
LIN {X 0,Y 530.343,Z 462.44,A -85,B 0,C 180,E1 4168.804,E2 4168.804} C_VEL
LIN {X 0,Y 530.303,Z 462.44,A -85,B 0,C 180,E1 4174.819,E2 4174.819} C_VEL
LIN {X 0,Y 530.301,Z 462.44,A -85,B 0,C 180,E1 4181.044,E2 4181.044} C_VEL
LIN {X 0,Y 530.285,Z 462.44,A -85,B 0,C 180,E1 4186.743,E2 4186.743} C_VEL
LIN {X 0,Y 530.361,Z 463.121,A -85,B 0,C 180,E1 4190.548,E2 4190.548} C_VEL
LIN {X 0,Y 546.255,Z 494.881,A -85,B 0,C 180,E1 4192.424,E2 4192.424} C_VEL
LIN {X 0,Y 545.197,Z 537.22,A -85,B 0,C 180,E1 4193.321,E2 4193.321} C_VEL
LIN {X 0,Y 543.416,Z 576.94,A -85,B 0,C 180,E1 4194.767,E2 4194.767} C_VEL
LIN {X 0,Y 541.179,Z 614.987,A -85,B 0,C 180,E1 4196.783,E2 4196.783} C_VEL
LIN {X 0,Y 538.493,Z 653.78,A -85,B 0,C 180,E1 4199.594,E2 4199.594} C_VEL
LIN {X 0,Y 535.92,Z 689.346,A -85,B 0,C 180,E1 4203.009,E2 4203.009} C_VEL
LIN {X 0,Y 533.882,Z 719.803,A -85,B 0,C 180,E1 4206.81,E2 4206.81} C_VEL
LIN {X 0,Y 532.365,Z 745.189,A -85,B 0,C 180,E1 4210.908,E2 4210.908} C_VEL
LIN {X 0,Y 531.575,Z 764.983,A -85,B 0,C 180,E1 4215.146,E2 4215.146} C_VEL
LIN {X 0,Y 531.137,Z 779.025,A -85,B 0,C 180,E1 4219.281,E2 4219.281} C_VEL
LIN {X 0,Y 531.058,Z 788.478,A -85,B 0,C 180,E1 4223.451,E2 4223.451} C_VEL
LIN {X 0,Y 531.007,Z 792.627,A -85,B 0,C 180,E1 4226.731,E2 4226.731} C_VEL
LIN {X 0,Y 531.011,Z 794,A -85,B 0,C 180,E1 4230,E2 4230} C_VEL
LIN {X 0,Y 530.961,Z 792.247,A -85,B 0,C 180,E1 4233.637,E2 4233.637} C_VEL
LIN {X 0,Y 531.125,Z 786.917,A -85,B 0,C 180,E1 4237.371,E2 4237.371} C_VEL
LIN {X 0,Y 531.221,Z 776.772,A -85,B 0,C 180,E1 4241.509,E2 4241.509} C_VEL
LIN {X 0,Y 531.73,Z 761.486,A -85,B 0,C 180,E1 4245.695,E2 4245.695} C_VEL
LIN {X 0,Y 532.636,Z 740.371,A -85,B 0,C 180,E1 4249.945,E2 4249.945} C_VEL
LIN {X 0,Y 534.157,Z 715.328,A -85,B 0,C 180,E1 4253.804,E2 4253.804} C_VEL
LIN {X 0,Y 536.281,Z 684.53,A -85,B 0,C 180,E1 4257.499,E2 4257.499} C_VEL
LIN {X 0,Y 538.759,Z 650.132,A -85,B 0,C 180,E1 4260.7,E2 4260.7} C_VEL
LIN {X 0,Y 541.252,Z 613.306,A -85,B 0,C 180,E1 4263.319,E2 4263.319} C_VEL
LIN {X 0,Y 543.622,Z 573.986,A -85,B 0,C 180,E1 4265.366,E2 4265.366} C_VEL
LIN {X 0,Y 545.409,Z 532.348,A -85,B 0,C 180,E1 4266.815,E2 4266.815} C_VEL
LIN {X 0,Y 545.958,Z 493.472,A -85,B 0,C 180,E1 4267.622,E2 4267.622} C_VEL
LIN {X 0,Y 530.361,Z 463.128,A -85,B 0,C 180,E1 4269.452,E2 4269.452} C_VEL
LIN {X 0,Y 530.307,Z 462.44,A -85,B 0,C 180,E1 4275.545,E2 4275.545} C_VEL
LIN {X 0,Y 530.306,Z 462.44,A -85,B 0,C 180,E1 4281.091,E2 4281.091} C_VEL
LIN {X 0,Y 530.276,Z 462.44,A -85,B 0,C 180,E1 4287.148,E2 4287.148} C_VEL
LIN {X 0,Y 530.407,Z 462.44,A -85,B 0,C 180,E1 4292.825,E2 4292.825} C_VEL
LIN {X 0,Y 530.554,Z 462.44,A -85,B 0,C 180,E1 4298.224,E2 4298.224} C_VEL
LIN {X 0,Y 530.601,Z 462.44,A -85,B 0,C 180,E1 4303.421,E2 4303.421} C_VEL
LIN {X 0,Y 530.629,Z 462.44,A -85,B 0,C 180,E1 4310.142,E2 4310.142} C_VEL
LIN {X 0,Y 530.806,Z 462.44,A -85,B 0,C 180,E1 4315.091,E2 4315.091} C_VEL
LIN {X 0,Y 530.824,Z 462.44,A -85,B 0,C 180,E1 4319.999,E2 4319.999} C_VEL
LIN {X 0,Y 530.759,Z 462.44,A -85,B 0,C 180,E1 4324.908,E2 4324.908} C_VEL
LIN {X 0,Y 530.694,Z 462.44,A -85,B 0,C 180,E1 4329.855,E2 4329.855} C_VEL
LIN {X 0,Y 530.608,Z 462.44,A -85,B 0,C 180,E1 4334.879,E2 4334.879} C_VEL
LIN {X 0,Y 530.529,Z 462.44,A -85,B 0,C 180,E1 4340.025,E2 4340.025} C_VEL
LIN {X 0,Y 530.419,Z 462.44,A -85,B 0,C 180,E1 4345.348,E2 4345.348} C_VEL
LIN {X 0,Y 530.328,Z 462.44,A -85,B 0,C 180,E1 4351.071,E2 4351.071} C_VEL
LIN {X 0,Y 530.346,Z 462.44,A -85,B 0,C 180,E1 4356.927,E2 4356.927} C_VEL
LIN {X 0,Y 530.119,Z 462.44,A -85,B 0,C 180,E1 4363.266,E2 4363.266} C_VEL
LIN {X 0,Y 530.242,Z 462.44,A -85,B 0,C 180,E1 4368.945,E2 4368.945} C_VEL
LIN {X 0,Y 530.542,Z 462.44,A -85,B 0,C 180,E1 4375.428,E2 4375.428} C_VEL
LIN {X 0,Y 530.554,Z 462.44,A -85,B 0,C 180,E1 4375.604,E2 4375.604} C_VEL
LIN {X 0,Y 542.552,Z 490.6,A -85,B 0,C 180,E1 4376.905,E2 4376.905} C_VEL
LIN {X 0,Y 542.111,Z 535.697,A -85,B 0,C 180,E1 4377.804,E2 4377.804} C_VEL
LIN {X 0,Y 540.615,Z 573.419,A -85,B 0,C 180,E1 4379.148,E2 4379.148} C_VEL
LIN {X 0,Y 538.834,Z 608.423,A -85,B 0,C 180,E1 4381.005,E2 4381.005} C_VEL
LIN {X 0,Y 536.705,Z 642.781,A -85,B 0,C 180,E1 4383.502,E2 4383.502} C_VEL
LIN {X 0,Y 534.784,Z 673.191,A -85,B 0,C 180,E1 4386.427,E2 4386.427} C_VEL
LIN {X 0,Y 533.144,Z 700.648,A -85,B 0,C 180,E1 4389.87,E2 4389.87} C_VEL
LIN {X 0,Y 532.025,Z 723.706,A -85,B 0,C 180,E1 4393.678,E2 4393.678} C_VEL
LIN {X 0,Y 531.364,Z 741.493,A -85,B 0,C 180,E1 4397.66,E2 4397.66} C_VEL
LIN {X 0,Y 531.165,Z 753.255,A -85,B 0,C 180,E1 4401.393,E2 4401.393} C_VEL
LIN {X 0,Y 531.028,Z 760.5,A -85,B 0,C 180,E1 4405.093,E2 4405.093} C_VEL
LIN {X 0,Y 530.971,Z 763.612,A -85,B 0,C 180,E1 4408.366,E2 4408.366} C_VEL
LIN {X 0,Y 531.073,Z 763.555,A -85,B 0,C 180,E1 4411.634,E2 4411.634} C_VEL
LIN {X 0,Y 531.1,Z 759.149,A -85,B 0,C 180,E1 4415.727,E2 4415.727} C_VEL
LIN {X 0,Y 531.218,Z 749.585,A -85,B 0,C 180,E1 4419.847,E2 4419.847} C_VEL
LIN {X 0,Y 531.648,Z 733.656,A -85,B 0,C 180,E1 4424.181,E2 4424.181} C_VEL
LIN {X 0,Y 532.58,Z 712.49,A -85,B 0,C 180,E1 4428.224,E2 4428.224} C_VEL
LIN {X 0,Y 534.018,Z 686.039,A -85,B 0,C 180,E1 4431.984,E2 4431.984} C_VEL
LIN {X 0,Y 535.837,Z 655.874,A -85,B 0,C 180,E1 4435.243,E2 4435.243} C_VEL
LIN {X 0,Y 537.972,Z 622.463,A -85,B 0,C 180,E1 4437.973,E2 4437.973} C_VEL
LIN {X 0,Y 539.988,Z 586.978,A -85,B 0,C 180,E1 4440.114,E2 4440.114} C_VEL
LIN {X 0,Y 541.589,Z 551.085,A -85,B 0,C 180,E1 4441.633,E2 4441.633} C_VEL
LIN {X 0,Y 542.661,Z 514.215,A -85,B 0,C 180,E1 4442.603,E2 4442.603} C_VEL
LIN {X 0,Y 542.233,Z 488.555,A -85,B 0,C 180,E1 4443.058,E2 4443.058} C_VEL
LIN {X 0,Y 530.332,Z 462.44,A -85,B 0,C 180,E1 4444.378,E2 4444.378} C_VEL
LIN {X 0,Y 530.299,Z 462.44,A -85,B 0,C 180,E1 4449.574,E2 4449.574} C_VEL
LIN {X 0,Y 530.249,Z 462.44,A -85,B 0,C 180,E1 4455.551,E2 4455.551} C_VEL
LIN {X 0,Y 530.226,Z 462.44,A -85,B 0,C 180,E1 4461.086,E2 4461.086} C_VEL
LIN {X 0,Y 530.254,Z 462.44,A -85,B 0,C 180,E1 4467.149,E2 4467.149} C_VEL
LIN {X 0,Y 530.385,Z 462.44,A -85,B 0,C 180,E1 4472.826,E2 4472.826} C_VEL
LIN {X 0,Y 530.549,Z 462.44,A -85,B 0,C 180,E1 4478.226,E2 4478.226} C_VEL
LIN {X 0,Y 530.66,Z 462.44,A -85,B 0,C 180,E1 4483.424,E2 4483.424} C_VEL
LIN {X 0,Y 530.682,Z 462.44,A -85,B 0,C 180,E1 4488.482,E2 4488.482} C_VEL
LIN {X 0,Y 530.705,Z 462.44,A -85,B 0,C 180,E1 4493.449,E2 4493.449} C_VEL
LIN {X 0,Y 530.757,Z 462.44,A -85,B 0,C 180,E1 4498.366,E2 4498.366} C_VEL
LIN {X 0,Y 530.773,Z 462.44,A -85,B 0,C 180,E1 4503.271,E2 4503.271} C_VEL
LIN {X 0,Y 530.659,Z 462.44,A -85,B 0,C 180,E1 4508.202,E2 4508.202} C_VEL
LIN {X 0,Y 530.579,Z 462.44,A -85,B 0,C 180,E1 4514.005,E2 4514.005} C_VEL
LIN {X 0,Y 530.529,Z 462.44,A -85,B 0,C 180,E1 4520.027,E2 4520.027} C_VEL
LIN {X 0,Y 530.513,Z 462.44,A -85,B 0,C 180,E1 4525.346,E2 4525.346} C_VEL
LIN {X 0,Y 530.343,Z 462.44,A -85,B 0,C 180,E1 4528.804,E2 4528.804} C_VEL
LIN {X 0,Y 527.809,Z 462.44,A -85,B 0,C 180,E1 4530.193,E2 4530.193} C_VEL
LIN {X 0,Y 522.428,Z 462.44,A -85,B 0,C 180,E1 4532.273,E2 4532.273} C_VEL
LIN {X 0,Y 522.352,Z 462.44,A -85,B 0,C 180,E1 4532.514,E2 4532.514} C_VEL
LIN {X 0,Y 522.36,Z 462.44,A -85,B 0,C 180,E1 4538.498,E2 4538.498} C_VEL
LIN {X 0,Y 522.421,Z 462.44,A -85,B 0,C 180,E1 4544.069,E2 4544.069} C_VEL
LIN {X 0,Y 522.356,Z 463.133,A -85,B 0,C 180,E1 4549.823,E2 4549.823} C_VEL
LIN {X 0,Y 539.95,Z 498.316,A -85,B 0,C 180,E1 4551.965,E2 4551.965} C_VEL
LIN {X 0,Y 538.614,Z 541.826,A -85,B 0,C 180,E1 4552.946,E2 4552.946} C_VEL
LIN {X 0,Y 536.555,Z 582.177,A -85,B 0,C 180,E1 4554.516,E2 4554.516} C_VEL
LIN {X 0,Y 534.069,Z 619.443,A -85,B 0,C 180,E1 4556.598,E2 4556.598} C_VEL
LIN {X 0,Y 531.323,Z 655.59,A -85,B 0,C 180,E1 4559.306,E2 4559.306} C_VEL
LIN {X 0,Y 528.525,Z 690.329,A -85,B 0,C 180,E1 4562.718,E2 4562.718} C_VEL
LIN {X 0,Y 526.318,Z 720.07,A -85,B 0,C 180,E1 4566.497,E2 4566.497} C_VEL
LIN {X 0,Y 524.674,Z 745.188,A -85,B 0,C 180,E1 4570.617,E2 4570.617} C_VEL
LIN {X 0,Y 523.748,Z 764.982,A -85,B 0,C 180,E1 4574.919,E2 4574.919} C_VEL
LIN {X 0,Y 523.263,Z 778.88,A -85,B 0,C 180,E1 4579.065,E2 4579.065} C_VEL
LIN {X 0,Y 523.154,Z 788.478,A -85,B 0,C 180,E1 4583.352,E2 4583.352} C_VEL
LIN {X 0,Y 523.127,Z 792.627,A -85,B 0,C 180,E1 4586.681,E2 4586.681} C_VEL
LIN {X 0,Y 523.121,Z 794,A -85,B 0,C 180,E1 4590,E2 4590} C_VEL
LIN {X 0,Y 523.12,Z 792.628,A -85,B 0,C 180,E1 4593.319,E2 4593.319} C_VEL
LIN {X 0,Y 523.242,Z 786.917,A -85,B 0,C 180,E1 4597.482,E2 4597.482} C_VEL
LIN {X 0,Y 523.346,Z 776.772,A -85,B 0,C 180,E1 4601.684,E2 4601.684} C_VEL
LIN {X 0,Y 523.912,Z 761.487,A -85,B 0,C 180,E1 4605.935,E2 4605.935} C_VEL
LIN {X 0,Y 524.974,Z 740.373,A -85,B 0,C 180,E1 4610.249,E2 4610.249} C_VEL
LIN {X 0,Y 526.703,Z 714.241,A -85,B 0,C 180,E1 4614.315,E2 4614.315} C_VEL
LIN {X 0,Y 529.01,Z 684.186,A -85,B 0,C 180,E1 4617.948,E2 4617.948} C_VEL
LIN {X 0,Y 531.741,Z 650.105,A -85,B 0,C 180,E1 4621.152,E2 4621.152} C_VEL
LIN {X 0,Y 534.528,Z 612.886,A -85,B 0,C 180,E1 4623.821,E2 4623.821} C_VEL
LIN {X 0,Y 537.153,Z 573.4,A -85,B 0,C 180,E1 4625.885,E2 4625.885} C_VEL
